// TwinCAT 3 PLC project tmo_motion
// Title: lcls-plc-tmo-motion
// Company: SLAC
// ProjectVersion: 0.0.0
// ProgramVersion: 3.1.4022.7
// CompilerDefines: K
// libraries:
//   LCLS General, * (SLAC)
//   lcls-twincat-common-components, * (SLAC)
//   lcls-twincat-motion, * (SLAC)
//   PMPS, * (SLAC - LCLS)
//   Tc2_MC2, * (Beckhoff Automation GmbH)
//   Tc2_SerialCom, * (Beckhoff Automation GmbH)
//   Tc2_Standard, * (Beckhoff Automation GmbH)
//   Tc2_System, * (Beckhoff Automation GmbH)
//   Tc3_Module, * (Beckhoff Automation GmbH)
// project tree:
//   DUTs/ ENUM_SolidAttenuator_States.TcDUT, ENUM_LaserCoupling_States.TcDUT, ENUM_Sample_Calibration_States.TcDUT, ENUM_ZonePlate_States.TcDUT, E_HomeState.TcDUT
//   GVLs/ GVL_PMPS.TcGVL, GVL_TcGVL.TcGVL, Main.TcGVL
//   / PlcTask.TcTTO (not stored)
//   POUs/ FB_SP_ZP.TcPOU, PRG_1_PlcTask.TcPOU, PRG_2_PMPS_PRE.TcPOU, PRG_3_PMPS_POST.TcPOU, PRG_4_LOG.TcPOU (not stored), PRG_AL1K4_L2SI.TcPOU, PRG_PA1K4_PF.TcPOU, PRG_IM2K4_PPM.TcPOU, PRG_IM3K4_PPM.TcPOU, PRG_IM4K4_PPM.TcPOU, PRG_IM5K4_PPM.TcPOU, PRG_IM6K4_PPM.TcPOU, PRG_LI1K4_IP1.TcPOU, PRG_LI2K4_IP1.TcPOU, PRG_PC5K4.TcPOU, PRG_PF1K4_WFS_TARGET.TcPOU, PRG_PF2K4_WFS_TARGET.TcPOU, PRG_SL1K4_SCATTER.TcPOU, PRG_SP1K4.TcPOU, PRG_ST4K4_TMO_TERM.TcPOU, PRG_ST5K4_TMO_TERM_FIXED.TcPOU, PRG_TM1K4.TcPOU, PRG_TM2K4.TcPOU
//   POUs/Sequence_Mover/ FB_SequenceMover2D.TcPOU
//   POUs/temp/ FB_SLITS.TcPOU, FB_SLITS_POWER.TcPOU, FB_SLITS_SCATTER.TcPOU, FB_ZonePlate_States.TcPOU, PRG_SL2K4_SCATTER.TcPOU
//   POUs/TM1K4/ ENUM_TM1K4_States.TcDUT, FB_TM1K4.TcPOU
//   POUs/TM2K4/ ENUM_TM2K4_States.TcDUT, FB_TM2K4.TcPOU
// real-time tasks:
//   TASK PlcTask: cycle T#10ms, priority 20, ADS port 350
// motion (NC):
//   TASK NC-Task 1 SAF: cycle T#2ms, priority 4, ADS port 501
//   TASK NC-Task 1 SVB: cycle T#10ms, priority 8, ADS port 511
//   AXIS Axis 1 AL1K4-L2SI-MMS (id 1)
//     Dynamic: AccelerationMaximum=200, DecelerationMaximum=200, Acceleration=200, Deceleration=200, Jerk=500, DelayTime=0.004
//     Velo: Maximum=10
//     TargetPosControl: Range=0.002, Time=2
//     OtherSettings: AllowMotionCmdToSlave=true
//     encoder EncType=29
//       EncPara: ScaleFactorNumerator=5e-05, Offset=-214686.941, MaxCount=#xffffffff, ReferenceSystem=1
//         SoftEndMinControl: Enable=true, Range=-108.74
//         SoftEndMaxControl: Enable=true, Range=-30
//         Inc: RefSoftSyncMask=#x0000ffff
//     drive DrvType=24
//       Analog: VeloReferenz=100, ScaleFactorActTorque=0.1
//       TimeComp: TaskDelayCycles=1
//     controller CtrType=2
//       CtrPara: PriorControlFactor=1
//         PosDiffControl: Range=1, Time=0.1
//         PID: PosKp=20, PosExtKp=1, PosExtVelo=0.1, DeadBandPosition=0.002
//         Observer: BandWidth=20
//   AXIS Axis 2 (id 2)
//     OtherSettings: AllowMotionCmdToSlave=true
//     encoder EncType=1
//     drive DrvType=5
//       Analog: ScaleFactorActTorque=0.1
//       TimeComp: TaskDelayCycles=1
//     controller CtrType=1
//       CtrPara: PriorControlFactor=1
//         Observer: BandWidth=20
//   AXIS Axis 3 (id 3)
//     OtherSettings: AllowMotionCmdToSlave=true
//     encoder EncType=1
//     drive DrvType=5
//       Analog: ScaleFactorActTorque=0.1
//       TimeComp: TaskDelayCycles=1
//     controller CtrType=1
//       CtrPara: PriorControlFactor=1
//         Observer: BandWidth=20
//   AXIS Axis 4 (id 4)
//     OtherSettings: AllowMotionCmdToSlave=true
//     encoder EncType=1
//     drive DrvType=5
//       Analog: ScaleFactorActTorque=0.1
//       TimeComp: TaskDelayCycles=1
//     controller CtrType=1
//       CtrPara: PriorControlFactor=1
//         Observer: BandWidth=20
//   AXIS Axis 5 (id 5)
//     OtherSettings: AllowMotionCmdToSlave=true
//     encoder EncType=1
//     drive DrvType=5
//       Analog: ScaleFactorActTorque=0.1
//       TimeComp: TaskDelayCycles=1
//     controller CtrType=1
//       CtrPara: PriorControlFactor=1
//         Observer: BandWidth=20
//   AXIS Axis 6 IM1K4-XTES-MMS (id 6)
//     Velo: Maximum=10
//     OtherSettings: AllowMotionCmdToSlave=true
//     encoder EncType=29
//       EncPara: ScaleFactorNumerator=5e-05, Offset=-398.1892, MaxCount=#x00400000, ReferenceSystem=1
//         SoftEndMinControl: Enable=true, Range=-90
//         SoftEndMaxControl: Enable=true
//         Inc: RefSoftSyncMask=#x00400000
//     drive DrvType=24
//       DrvPara: Inverse=true
//         Analog: VeloReferenz=50, ScaleFactorActTorque=0.1
//         TimeComp: TaskDelayCycles=1
//     controller CtrType=2
//       CtrPara: PriorControlFactor=1
//         PosDiffControl: Range=1
//         PID: PosKp=20, PosExtKp=20, DeadBandPosition=0.001
//         Observer: BandWidth=20
//   AXIS Axis 7 IM1K4-XTES-CLZ (id 7)
//     General: UnitName=%
//     Velo: Maximum=10
//     OtherSettings: AllowMotionCmdToSlave=true
//     encoder EncType=4
//       EncPara: ScaleFactorNumerator=0.003, MaxCount=#x0000ffff
//         SoftEndMinControl: Enable=true, Range=-100
//         SoftEndMaxControl: Enable=true, Range=100
//         Inc: RefSoftSyncMask=#x0000ffff
//     drive DrvType=23
//       DrvPara: Inverse=true
//         Analog: VeloReferenz=33, ScaleFactorActTorque=0.1
//         TimeComp: TaskDelayCycles=1
//     controller CtrType=2
//       CtrPara: PriorControlFactor=1
//         PosDiffControl: Range=1
//         PID: PosKp=20, PosExtKp=20, DeadBandPosition=0.1
//         Observer: BandWidth=20
//   AXIS Axis 8 IM1K4-XTES-CLF (id 8)
//     General: UnitName=%
//     Velo: Maximum=10
//     OtherSettings: AllowMotionCmdToSlave=true
//     encoder EncType=4
//       EncPara: ScaleFactorNumerator=0.008, MaxCount=#x0000ffff
//         SoftEndMinControl: Enable=true, Range=-100
//         SoftEndMaxControl: Enable=true, Range=100
//         Inc: RefSoftSyncMask=#x0000ffff
//     drive DrvType=23
//       DrvPara: Inverse=true
//         Analog: VeloReferenz=70, ScaleFactorActTorque=0.1
//         TimeComp: TaskDelayCycles=1
//     controller CtrType=2
//       CtrPara: PriorControlFactor=1
//         PosDiffControl: Range=1
//         PID: PosKp=20, PosExtKp=20, DeadBandPosition=0.1
//         Observer: BandWidth=20
//   AXIS Axis 9 IM2K4-PPM-MMS (id 9)
//     Dynamic: AccelerationMaximum=200, DecelerationMaximum=200, Acceleration=200, Deceleration=200, Jerk=1000, DelayTime=0.004
//     Velo: Maximum=65
//     MotionControl: Enable=true, Range=0.0005, Time=1
//     TargetPosControl: Range=0.01, Time=1
//     OtherSettings: AllowMotionCmdToSlave=true
//     encoder EncType=29
//       EncPara: ScaleFactorNumerator=5e-05, Offset=-358.0066, MaxCount=#x00400000, ReferenceSystem=1
//         SoftEndMinControl: Enable=true, Range=-100.57
//         SoftEndMaxControl: Enable=true, Range=-7.67
//         Inc: RefSoftSyncMask=#x00400000
//     drive DrvType=24
//       Analog: VeloReferenz=100, ScaleFactorActTorque=0.1
//       TimeComp: TaskDelayCycles=1
//     controller CtrType=2
//       CtrPara: PriorControlFactor=1
//         PosDiffControl: Range=10, Time=0.1
//         PID: PosKp=10, PosExtKp=0.01, PosExtVelo=0.0005, DeadBandPosition=0.0001
//         Observer: BandWidth=20
//   AXIS SL1K4-BOTTOM-M10 (id 10)
//     Velo: RefSearch=0.2, RefSync=0.05, Maximum=2.2
//     OtherSettings: AllowMotionCmdToSlave=true
//     encoder EncType=4
//       EncPara: MaxCount=#x0000ffff
//         SoftEndMinControl: Enable=true, Range=-31.51
//         SoftEndMaxControl: Enable=true
//         Inc: RefSoftSyncMask=#x0000ffff
//     drive DrvType=24
//       Analog: VeloReferenz=2, ScaleFactorActTorque=0.1
//       TimeComp: TaskDelayCycles=1
//     controller CtrType=1
//       CtrPara: PriorControlFactor=1
//         PosDiffControl: Range=0.05
//         Observer: BandWidth=20
//   AXIS SL1K4-TOP-M11 (id 11)
//     Velo: RefSearch=0.2, RefSync=0.05, Maximum=2.2
//     OtherSettings: AllowMotionCmdToSlave=true
//     encoder EncType=4
//       EncPara: Inverse=true, MaxCount=#x0000ffff
//         SoftEndMinControl: Enable=true, Range=-31.99
//         SoftEndMaxControl: Enable=true
//         Inc: RefSoftSyncMask=#x0000ffff
//     drive DrvType=24
//       Analog: VeloReferenz=2, ScaleFactorActTorque=0.1
//       TimeComp: TaskDelayCycles=1
//     controller CtrType=1
//       CtrPara: PriorControlFactor=1
//         PosDiffControl: Range=0.05
//         Observer: BandWidth=20
//   AXIS SL1K4-NORTH-M12 (id 12)
//     Velo: RefSearch=0.2, RefSync=0.05, Maximum=2.2
//     OtherSettings: AllowMotionCmdToSlave=true
//     encoder EncType=4
//       EncPara: Inverse=true, MaxCount=#x0000ffff
//         SoftEndMinControl: Enable=true, Range=-31.5
//         SoftEndMaxControl: Enable=true
//         Inc: RefSoftSyncMask=#x0000ffff
//     drive DrvType=24
//       Analog: VeloReferenz=2, ScaleFactorActTorque=0.1
//       TimeComp: TaskDelayCycles=1
//     controller CtrType=1
//       CtrPara: PriorControlFactor=1
//         PosDiffControl: Range=0.05
//         Observer: BandWidth=20
//   AXIS SL1K4-SOUTH-M13 (id 13)
//     Velo: RefSearch=0.2, RefSync=0.05, Maximum=2.2
//     OtherSettings: AllowMotionCmdToSlave=true
//     encoder EncType=4
//       EncPara: MaxCount=#x0000ffff
//         SoftEndMinControl: Enable=true, Range=-30.29
//         SoftEndMaxControl: Enable=true
//         Inc: RefSoftSyncMask=#x0000ffff
//     drive DrvType=24
//       Analog: VeloReferenz=2, ScaleFactorActTorque=0.1
//       TimeComp: TaskDelayCycles=1
//     controller CtrType=1
//       CtrPara: PriorControlFactor=1
//         PosDiffControl: Range=0.05
//         Observer: BandWidth=20
//   AXIS ST1K4-TEST (id 14)
//     Velo: RefSearch=5, RefSync=5, SlowManual=1, FastManual=5, Maximum=50
//     OtherSettings: AllowMotionCmdToSlave=true
//     encoder EncType=4
//       EncPara: ScaleFactorNumerator=0.000390625, Inverse=true, MaxCount=#x0000ffff
//         Inc: RefSoftSyncMask=#x0000ffff
//     drive DrvType=24
//       DrvPara: Inverse=true
//         Analog: VeloReferenz=50
//         TimeComp: TaskDelayCycles=1
//     controller CtrType=1
//       CtrPara: PriorControlFactor=1
//         PosDiffControl: Enable=false, Range=0.05
//         Observer: BandWidth=20
//   AXIS Axis 15 IM3K4-PPM-MMS (id 15)
//     Dynamic: AccelerationMaximum=200, DecelerationMaximum=200, Acceleration=200, Deceleration=200, Jerk=1000, DelayTime=0.004
//     Velo: Maximum=65
//     MotionControl: Enable=true, Range=0.0005, Time=1
//     TargetPosControl: Range=0.01, Time=1
//     OtherSettings: AllowMotionCmdToSlave=true
//     encoder EncType=29
//       EncPara: ScaleFactorNumerator=5e-05, Offset=-358.0066, MaxCount=#x00400000, ReferenceSystem=1
//         SoftEndMinControl: Enable=true, Range=-97.98
//         SoftEndMaxControl: Enable=true, Range=-5.69
//     drive DrvType=24
//       Analog: VeloReferenz=100, ScaleFactorActTorque=0.1
//       TimeComp: TaskDelayCycles=1
//     controller CtrType=2
//       CtrPara: PriorControlFactor=1
//         PosDiffControl: Range=10, Time=0.1
//         PID: PosKp=10, PosExtKp=0.01, PosExtVelo=0.0005, DeadBandPosition=0.0001
//         Observer: BandWidth=20
//   AXIS Axis 16 IM4K4-PPM-MMS (id 16)
//     Dynamic: AccelerationMaximum=200, DecelerationMaximum=200, Acceleration=200, Deceleration=200, Jerk=1000, DelayTime=0.004
//     Velo: Maximum=65
//     MotionControl: Enable=true, Range=0.0005, Time=1
//     TargetPosControl: Range=0.01, Time=1
//     OtherSettings: AllowMotionCmdToSlave=true
//     encoder EncType=29
//       EncPara: ScaleFactorNumerator=5e-05, Offset=-358.0066, MaxCount=#x00400000, ReferenceSystem=1
//         SoftEndMinControl: Enable=true, Range=-99.53
//         SoftEndMaxControl: Enable=true, Range=-8.43
//     drive DrvType=24
//       Analog: VeloReferenz=100, ScaleFactorActTorque=0.1
//       TimeComp: TaskDelayCycles=1
//     controller CtrType=2
//       CtrPara: PriorControlFactor=1
//         PosDiffControl: Range=10, Time=0.1
//         PID: PosKp=10, PosExtKp=0.01, PosExtVelo=0.0005, DeadBandPosition=0.0001
//         Observer: BandWidth=20
//   AXIS Axis 17 IM5K4-PPM-MMS (id 17)
//     Dynamic: AccelerationMaximum=200, DecelerationMaximum=200, Acceleration=200, Deceleration=200, Jerk=1000, DelayTime=0.004
//     Velo: Maximum=65
//     MotionControl: Enable=true, Range=0.0005, Time=1
//     TargetPosControl: Range=0.01, Time=1
//     OtherSettings: AllowMotionCmdToSlave=true
//     encoder EncType=29
//       EncPara: ScaleFactorNumerator=5e-05, Offset=-358.0066, MaxCount=#x00400000, ReferenceSystem=1
//         SoftEndMinControl: Enable=true, Range=-97.47
//         SoftEndMaxControl: Enable=true, Range=-4.42
//     drive DrvType=24
//       Analog: VeloReferenz=100, ScaleFactorActTorque=0.1
//       TimeComp: TaskDelayCycles=1
//     controller CtrType=2
//       CtrPara: PriorControlFactor=1
//         PosDiffControl: Range=10, Time=0.1
//         PID: PosKp=10, PosExtKp=0.01, PosExtVelo=0.0005, DeadBandPosition=0.0001
//         Observer: BandWidth=20
//   AXIS Axis 18 PF1K4-WFS_TARGET-MMS-Y (id 18)
//     Dynamic: AccelerationMaximum=200, DecelerationMaximum=200, Acceleration=10, Deceleration=10, Jerk=500, DelayTime=0.004
//     Velo: Maximum=20
//     TargetPosControl: Range=0.002, Time=2
//     OtherSettings: AllowMotionCmdToSlave=true
//     encoder EncType=29
//       EncPara: ScaleFactorNumerator=5e-05, Offset=-358.0066, MaxCount=#x00400000, ReferenceSystem=1
//         SoftEndMinControl: Enable=true, Range=-99.33
//         SoftEndMaxControl: Enable=true, Range=-9.97777
//     drive DrvType=24
//       Analog: VeloReferenz=100, ScaleFactorActTorque=0.1
//       TimeComp: TaskDelayCycles=1
//     controller CtrType=2
//       CtrPara: PriorControlFactor=1
//         PosDiffControl: Range=1
//         PID: PosKp=20, PosExtKp=1, PosExtVelo=0.1, DeadBandPosition=0.002
//         Observer: BandWidth=20
//   AXIS Axis 19 PF1K4-WFS_TARGET-MMS-Z (id 19)
//     Dynamic: AccelerationMaximum=200, DecelerationMaximum=200, Acceleration=10, Deceleration=50, Jerk=500
//     Velo: Maximum=5
//     OtherSettings: AllowMotionCmdToSlave=true
//     encoder EncType=29
//       EncPara: ScaleFactorNumerator=5e-05, MaxCount=#xffffffff
//         SoftEndMinControl: Enable=true, Range=12
//         SoftEndMaxControl: Enable=true, Range=54
//         Inc: RefSoftSyncMask=#x0000ffff
//     drive DrvType=24
//       Analog: VeloReferenz=15.875, TorqueSetpointScale=10, ScaleFactorActTorque=0.1
//       TimeComp: TaskDelayCycles=1
//     controller CtrType=1
//       CtrPara: PriorControlFactor=1
//         PosDiffControl: Range=1
//         Observer: BandWidth=20
//   AXIS Axis 20 LI1K4-IP1-MMS (id 20)
//     Dynamic: AccelerationMaximum=200, DecelerationMaximum=200, Acceleration=200, Deceleration=200, Jerk=500, DelayTime=0.004
//     Velo: Maximum=65
//     TargetPosControl: Range=0.002, Time=2
//     OtherSettings: AllowMotionCmdToSlave=true
//     encoder EncType=29
//       EncPara: ScaleFactorNumerator=5e-05, Offset=-358.0066, MaxCount=#x00400000, ReferenceSystem=1
//         SoftEndMinControl: Enable=true, Range=-107.43
//         SoftEndMaxControl: Enable=true, Range=1.35
//     drive DrvType=24
//       Analog: VeloReferenz=100, ScaleFactorActTorque=0.1
//       TimeComp: TaskDelayCycles=1
//     controller CtrType=2
//       CtrPara: PriorControlFactor=1
//         PosDiffControl: Range=1
//         PID: PosKp=20, PosExtKp=1, PosExtVelo=0.1, DeadBandPosition=0.002
//         Observer: BandWidth=20
//   AXIS Axis 21 TM1K4-MMS-Y (id 21)
//     Dynamic: AccelerationMaximum=200, DecelerationMaximum=200, Acceleration=10, Deceleration=10, Jerk=500, DelayTime=0.004
//     Velo: Maximum=20
//     TargetPosControl: Range=0.002, Time=2
//     OtherSettings: AllowMotionCmdToSlave=true
//     encoder EncType=29
//       EncPara: ScaleFactorNumerator=5e-05, Offset=-358.0066, MaxCount=#x00400000, ReferenceSystem=1
//         SoftEndMinControl: Enable=true, Range=-103.65
//         SoftEndMaxControl: Enable=true, Range=1.41
//     drive DrvType=24
//       Analog: VeloReferenz=100, ScaleFactorActTorque=0.1
//       TimeComp: TaskDelayCycles=1
//     controller CtrType=2
//       CtrPara: PriorControlFactor=1
//         PosDiffControl: Enable=false, Range=1
//         PID: PosKp=20, PosExtKp=1, PosExtVelo=0.1, DeadBandPosition=0.002
//         Observer: BandWidth=20
//   AXIS Axis 22 TM1K4-MMS-X (id 22)
//     Dynamic: AccelerationMaximum=200, DecelerationMaximum=200, Acceleration=10, Deceleration=50, Jerk=500
//     Velo: Maximum=5
//     OtherSettings: AllowMotionCmdToSlave=true
//     encoder EncType=29
//       EncPara: ScaleFactorNumerator=5e-05, MaxCount=#xffffffff
//         SoftEndMinControl: Enable=true, Range=12
//         SoftEndMaxControl: Enable=true, Range=54
//         Inc: RefSoftSyncMask=#x0000ffff
//     drive DrvType=24
//       Analog: VeloReferenz=15.875, TorqueSetpointScale=10, ScaleFactorActTorque=0.1
//       TimeComp: TaskDelayCycles=1
//     controller CtrType=1
//       CtrPara: PriorControlFactor=1
//         PosDiffControl: Range=1
//         Observer: BandWidth=20
//   AXIS SL2K4-BOTTOM-M23 (id 23) // C:\Github\lcls-plc-tmo-motion\plc-tmo-motion\_Config\NC\Axes\SL2K4-BOTTOM-M23.xti
//     Velo: RefSearch=0.2, RefSync=0.05, Maximum=2.2
//     OtherSettings: AllowMotionCmdToSlave=true
//     encoder EncType=4
//       EncPara: MaxCount=#x0000ffff
//         SoftEndMinControl: Enable=true, Range=-30.61
//         SoftEndMaxControl: Enable=true
//         Inc: RefSoftSyncMask=#x0000ffff
//     drive DrvType=24
//       Analog: VeloReferenz=2, ScaleFactorActTorque=0.1
//       TimeComp: TaskDelayCycles=1
//     controller CtrType=1
//       CtrPara: PriorControlFactor=1
//         Observer: BandWidth=20
//   AXIS SL2K4-TOP-M24 (id 24) // C:\Github\lcls-plc-tmo-motion\plc-tmo-motion\_Config\NC\Axes\SL2K4-TOP-M24.xti
//     Velo: RefSearch=0.2, RefSync=0.05, Maximum=2.2
//     PositionAreaControl: Range=0.5
//     TargetPosControl: Range=0.1
//     OtherSettings: AllowMotionCmdToSlave=true
//     encoder EncType=4
//       EncPara: Inverse=true, MaxCount=#x0000ffff
//         SoftEndMinControl: Enable=true, Range=-30.91
//         SoftEndMaxControl: Enable=true
//         Inc: RefSoftSyncMask=#x0000ffff
//     drive DrvType=24
//       Analog: VeloReferenz=2, ScaleFactorActTorque=0.1
//       TimeComp: TaskDelayCycles=1
//     controller CtrType=1
//       CtrPara: PriorControlFactor=1
//         PosDiffControl: Range=0.5
//         Observer: BandWidth=20
//   AXIS SL2K4-NORTH-M25 (id 25) // C:\Github\lcls-plc-tmo-motion\plc-tmo-motion\_Config\NC\Axes\SL2K4-NORTH-M25.xti
//     Velo: RefSearch=0.2, RefSync=0.05, Maximum=2.2
//     OtherSettings: AllowMotionCmdToSlave=true
//     encoder EncType=4
//       EncPara: Inverse=true, MaxCount=#x0000ffff
//         SoftEndMinControl: Enable=true, Range=-30.81
//         SoftEndMaxControl: Enable=true
//         Inc: RefSoftSyncMask=#x0000ffff
//     drive DrvType=24
//       Analog: VeloReferenz=2, ScaleFactorActTorque=0.1
//       TimeComp: TaskDelayCycles=1
//     controller CtrType=1
//       CtrPara: PriorControlFactor=1
//         Observer: BandWidth=20
//   AXIS SL2K4-SOUTH-M26 (id 26) // C:\Github\lcls-plc-tmo-motion\plc-tmo-motion\_Config\NC\Axes\SL2K4-SOUTH-M26.xti
//     Velo: RefSearch=0.2, RefSync=0.05, Maximum=2.2
//     OtherSettings: AllowMotionCmdToSlave=true
//     encoder EncType=4
//       EncPara: MaxCount=#x0000ffff
//         SoftEndMinControl: Enable=true, Range=-30.52
//         SoftEndMaxControl: Enable=true
//         Inc: RefSoftSyncMask=#x0000ffff
//     drive DrvType=24
//       Analog: VeloReferenz=2, ScaleFactorActTorque=0.1
//       TimeComp: TaskDelayCycles=1
//     controller CtrType=1
//       CtrPara: PriorControlFactor=1
//         Observer: BandWidth=20
//   AXIS Axis 30 TM2K4-MMS-Y (id 30)
//     Dynamic: AccelerationMaximum=200, DecelerationMaximum=200, Acceleration=10, Deceleration=10, Jerk=500, DelayTime=0.004
//     Velo: Maximum=20
//     TargetPosControl: Range=0.002, Time=2
//     OtherSettings: AllowMotionCmdToSlave=true
//     encoder EncType=29
//       EncPara: ScaleFactorNumerator=5e-05, Offset=-358.0066, MaxCount=#x00400000, ReferenceSystem=1
//         SoftEndMinControl: Enable=true, Range=-103
//         SoftEndMaxControl: Enable=true, Range=2.2
//     drive DrvType=24
//       Analog: VeloReferenz=100, ScaleFactorActTorque=0.1
//       TimeComp: TaskDelayCycles=1
//     controller CtrType=2
//       CtrPara: PriorControlFactor=1
//         PosDiffControl: Range=1
//         PID: PosKp=20, PosExtKp=1, PosExtVelo=0.1, DeadBandPosition=0.002
//         Observer: BandWidth=20
//   AXIS Axis 31 TM2K4-MMS-X (id 31)
//     Dynamic: AccelerationMaximum=200, DecelerationMaximum=200, Acceleration=10, Deceleration=50, Jerk=500
//     Velo: Maximum=5
//     OtherSettings: AllowMotionCmdToSlave=true
//     encoder EncType=29
//       EncPara: ScaleFactorNumerator=5e-05, MaxCount=#x00400000, ReferenceSystem=1
//         SoftEndMinControl: Enable=true, Range=7
//         SoftEndMaxControl: Enable=true, Range=11
//     drive DrvType=24
//       Analog: VeloReferenz=15.875, ScaleFactorActTorque=0.1
//       TimeComp: TaskDelayCycles=1
//     controller CtrType=1
//       CtrPara: PriorControlFactor=1
//         PosDiffControl: Range=0.2
//         Observer: BandWidth=20
//   AXIS Axis 27 IM6K4-PPM-MMS (id 27)
//     Dynamic: AccelerationMaximum=200, DecelerationMaximum=200, Acceleration=200, Deceleration=200, Jerk=500, DelayTime=0.004
//     Velo: Maximum=65
//     TargetPosControl: Range=0.002, Time=2
//     OtherSettings: AllowMotionCmdToSlave=true
//     encoder EncType=29
//       EncPara: ScaleFactorNumerator=5e-05, Offset=-358.0066, MaxCount=#x00400000, ReferenceSystem=1
//         SoftEndMinControl: Enable=true, Range=-97
//         SoftEndMaxControl: Enable=true, Range=-6.5
//     drive DrvType=24
//       Analog: VeloReferenz=100, ScaleFactorActTorque=0.1
//       TimeComp: TaskDelayCycles=1
//     controller CtrType=2
//       CtrPara: PriorControlFactor=1
//         PosDiffControl: Range=10, Time=0.1
//         PID: PosKp=10, PosExtKp=0.01, PosExtVelo=0.0005, DeadBandPosition=0.0001
//         Observer: BandWidth=20
//   AXIS Axis 28 PF2K4-WFS_TARGET-MMS-Y (id 28)
//     Dynamic: AccelerationMaximum=200, DecelerationMaximum=200, Acceleration=10, Deceleration=10, Jerk=500, DelayTime=0.004
//     Velo: Maximum=20
//     TargetPosControl: Range=0.002, Time=2
//     OtherSettings: AllowMotionCmdToSlave=true
//     encoder EncType=29
//       EncPara: ScaleFactorNumerator=5e-05, Offset=-358.065999999999, MaxCount=#x00400000, ReferenceSystem=1
//         SoftEndMinControl: Enable=true, Range=-103
//         SoftEndMaxControl: Enable=true, Range=-9.71
//     drive DrvType=24
//       Analog: VeloReferenz=100, ScaleFactorActTorque=0.1
//       TimeComp: TaskDelayCycles=1
//     controller CtrType=2
//       CtrPara: PriorControlFactor=1
//         PosDiffControl: Range=1
//         PID: PosKp=20, PosExtKp=1, PosExtVelo=0.1, DeadBandPosition=0.002
//         Observer: BandWidth=20
//   AXIS Axis 29 PF2K4-WFS_TARGET-MMS-Z (id 29)
//     Dynamic: AccelerationMaximum=200, DecelerationMaximum=200, Acceleration=10, Deceleration=50, Jerk=500
//     Velo: Maximum=5
//     OtherSettings: AllowMotionCmdToSlave=true
//     encoder EncType=29
//       EncPara: ScaleFactorNumerator=5e-05, MaxCount=#x00400000, ReferenceSystem=1
//         SoftEndMinControl: Enable=true, Range=17
//         SoftEndMaxControl: Enable=true, Range=50
//     drive DrvType=24
//       DrvPara: Inverse=true
//         Analog: VeloReferenz=15.875, ScaleFactorActTorque=0.1
//         TimeComp: TaskDelayCycles=1
//     controller CtrType=1
//       CtrPara: PriorControlFactor=1
//         PosDiffControl: Range=1
//         Observer: BandWidth=20
//   AXIS LensX (id 32)
//     Dynamic: Acceleration=2, Deceleration=2
//     Velo: SlowManual=0.1, FastManual=1, Maximum=1
//     OtherSettings: AllowMotionCmdToSlave=true, PulseDistancePos=0.5, PulseDistanceNeg=0.5
//     encoder EncType=4
//       EncPara: ScaleFactorNumerator=3.90625e-05, MaxCount=#x0000ffff
//         Inc: RefSoftSyncMask=#x0000ffff
//     drive DrvType=24
//       Analog: VeloReferenz=4.5, ScaleFactorActTorque=0.1
//       TimeComp: TaskDelayCycles=1
//     controller CtrType=2
//       CtrPara: PriorControlFactor=1
//         PosDiffControl: Range=1
//         Observer: BandWidth=20
//   AXIS FoilX (id 33)
//     Dynamic: Acceleration=2, Deceleration=2
//     Velo: SlowManual=0.1, FastManual=1, Maximum=27
//     PositionAreaControl: Range=0.1
//     TargetPosControl: Range=0.1
//     OtherSettings: AllowMotionCmdToSlave=true, PulseDistancePos=0.5, PulseDistanceNeg=0.5
//     encoder EncType=29
//       EncPara: ScaleFactorNumerator=5e-05, MaxCount=#xffffffff
//         Inc: RefSoftSyncMask=#x0000ffff
//     drive DrvType=24
//       DrvPara: Inverse=true
//         Analog: VeloReferenz=25.4, ScaleFactorActTorque=0.1
//         TimeComp: TaskDelayCycles=1
//     controller CtrType=2
//       CtrPara: PriorControlFactor=1
//         PosDiffControl: Range=0.8
//         Observer: BandWidth=20
//   AXIS ZonePlateX (id 34)
//     Dynamic: Acceleration=2, Deceleration=2
//     Velo: SlowManual=0.1, FastManual=1, Maximum=5
//     TargetPosControl: Range=0.03, Time=0.1
//     OtherSettings: AllowMotionCmdToSlave=true, PulseDistancePos=0.5, PulseDistanceNeg=0.5
//     encoder EncType=29
//       EncPara: ScaleFactorNumerator=5e-05, MaxCount=#xffffffff
//         SoftEndMinControl: Enable=true
//         SoftEndMaxControl: Enable=true, Range=125.6
//         Inc: RefSoftSyncMask=#x0000ffff
//     drive DrvType=24
//       DrvPara: Inverse=true
//         Analog: VeloReferenz=13.2, ScaleFactorActTorque=0.1
//         TimeComp: TaskDelayCycles=1
//     controller CtrType=2
//       CtrPara: PriorControlFactor=1
//         PosDiffControl: Range=1
//         PID: PosKp=2
//         Observer: BandWidth=20
//   AXIS ZonePlateY (id 35)
//     Dynamic: Acceleration=2, Deceleration=2
//     Velo: SlowManual=0.1, FastManual=1, Maximum=5
//     OtherSettings: AllowMotionCmdToSlave=true, PulseDistancePos=0.5, PulseDistanceNeg=0.5
//     encoder EncType=29
//       EncPara: ScaleFactorNumerator=5e-05, Offset=-214733.3875, MaxCount=#xffffffff
//         SoftEndMinControl: Enable=true, Range=-10.6
//         SoftEndMaxControl: Enable=true, Range=3.8
//         Inc: RefSoftSyncMask=#x0000ffff
//     drive DrvType=24
//       Analog: VeloReferenz=6, ScaleFactorActTorque=0.1
//       TimeComp: TaskDelayCycles=1
//     controller CtrType=2
//       CtrPara: PriorControlFactor=1
//         PosDiffControl: Range=0.8, Time=0.1
//         Observer: BandWidth=20
//   AXIS ZonePlateZ (id 36)
//     Dynamic: Acceleration=2, Deceleration=2
//     Velo: SlowManual=0.1, FastManual=1, Maximum=5
//     TargetPosControl: Range=0.3
//     OtherSettings: AllowMotionCmdToSlave=true, PulseDistancePos=0.5, PulseDistanceNeg=0.5
//     encoder EncType=29
//       EncPara: ScaleFactorNumerator=5e-05, ScaleFactorDenominator=1.6, Offset=-134207.665, MaxCount=#xffffffff
//         SoftEndMinControl: Enable=true, Range=-1
//         SoftEndMaxControl: Enable=true, Range=2
//         Inc: RefSoftSyncMask=#x0000ffff
//     drive DrvType=24
//       Analog: VeloReferenz=6.25, ScaleFactorActTorque=0.1
//       TimeComp: TaskDelayCycles=1
//     controller CtrType=2
//       CtrPara: PriorControlFactor=1
//         PosDiffControl: Range=1
//         Observer: BandWidth=20
//   AXIS YagX (id 37)
//     Dynamic: Acceleration=2, Deceleration=2
//     Velo: SlowManual=0.1, FastManual=1, Maximum=1
//     OtherSettings: AllowMotionCmdToSlave=true, PulseDistancePos=0.5, PulseDistanceNeg=0.5
//     encoder EncType=29
//       EncPara: ScaleFactorNumerator=5e-05, Offset=128, Inverse=true, MaxCount=#xffffffff, MaxCountHighDWord=#x0000001f
//         Inc: RefSoftSyncMask=#x0000ffff
//     drive DrvType=24
//       Analog: VeloReferenz=10, ScaleFactorActTorque=0.1
//       TimeComp: TaskDelayCycles=1
//     controller CtrType=2
//       CtrPara: PriorControlFactor=1
//         PosDiffControl: Range=1
//         Observer: BandWidth=20
//   AXIS YagY (id 38)
//     Dynamic: Acceleration=2, Deceleration=2
//     Velo: SlowManual=0.1, FastManual=1, Maximum=1
//     OtherSettings: AllowMotionCmdToSlave=true, PulseDistancePos=0.5, PulseDistanceNeg=0.5
//     encoder EncType=4
//       EncPara: ScaleFactorNumerator=7.8125e-05, MaxCount=#x0000ffff
//         Inc: RefSoftSyncMask=#x0000ffff
//     drive DrvType=24
//       Analog: VeloReferenz=10, ScaleFactorActTorque=0.1
//       TimeComp: TaskDelayCycles=1
//     controller CtrType=2
//       CtrPara: PriorControlFactor=1
//         PosDiffControl: Range=1
//         Observer: BandWidth=20
//   AXIS YagZ (id 39)
//     Dynamic: Acceleration=2, Deceleration=2
//     Velo: SlowManual=0.1, FastManual=1, Maximum=1
//     OtherSettings: AllowMotionCmdToSlave=true, PulseDistancePos=0.5, PulseDistanceNeg=0.5
//     encoder EncType=29
//       EncPara: ScaleFactorNumerator=5e-05, Offset=172, Inverse=true, MaxCount=#xffffffff, MaxCountHighDWord=#x0000001f
//         Inc: RefSoftSyncMask=#x0000ffff
//     drive DrvType=24
//       Analog: VeloReferenz=12.7, ScaleFactorActTorque=0.1
//       TimeComp: TaskDelayCycles=1
//     controller CtrType=2
//       CtrPara: PriorControlFactor=1
//         PosDiffControl: Range=1
//         Observer: BandWidth=20
//   AXIS YagTheta (id 40)
//     Dynamic: Acceleration=2, Deceleration=2
//     Velo: SlowManual=0.1, FastManual=1, Maximum=1
//     TargetPosControl: Range=0.001, Time=0.8
//     OtherSettings: AllowMotionCmdToSlave=true, PulseDistancePos=0.5, PulseDistanceNeg=0.5
//     encoder EncType=4
//       EncPara: ScaleFactorNumerator=1.171875e-05, ScaleFactorDenominator=0.036667, MaxCount=#x0000ffff
//         Inc: RefSoftSyncMask=#x0000ffff
//     drive DrvType=24
//       Analog: VeloReferenz=409.0905372, ScaleFactorActTorque=0.1
//       TimeComp: TaskDelayCycles=1
//     controller CtrType=2
//       CtrPara: PriorControlFactor=1
//         PosDiffControl: Range=1
//         PID: PosKp=5, DeadBandPosition=0.001
//         Observer: BandWidth=20
//   AXIS Thorlabs1 (id 41)
//     Dynamic: AccelerationMaximum=10, DecelerationMaximum=10, Acceleration=5, Deceleration=5
//     Velo: Maximum=2
//     OtherSettings: AllowMotionCmdToSlave=true
//     encoder EncType=4
//       EncPara: ScaleFactorNumerator=1.593130056e-05, MaxCount=#x0000ffff
//         Inc: RefSoftSyncMask=#x0000ffff
//     drive DrvType=24
//       Analog: VeloReferenz=2.039206472, ScaleFactorActTorque=0.1
//       TimeComp: TaskDelayCycles=1
//     controller CtrType=1
//       CtrPara: PriorControlFactor=1
//         PID: PosKp=0
//         Observer: BandWidth=20
//   AXIS Thorlabs2 (id 42)
//     Dynamic: AccelerationMaximum=10, DecelerationMaximum=10, Acceleration=5, Deceleration=5
//     Velo: Maximum=2
//     OtherSettings: AllowMotionCmdToSlave=true
//     encoder EncType=4
//       EncPara: ScaleFactorNumerator=1.593130056e-05, MaxCount=#x0000ffff
//         Inc: RefSoftSyncMask=#x0000ffff
//     drive DrvType=24
//       Analog: VeloReferenz=2.039206472, ScaleFactorActTorque=0.1
//       TimeComp: TaskDelayCycles=1
//     controller CtrType=1
//       CtrPara: PriorControlFactor=1
//         PID: PosKp=0
//         Observer: BandWidth=20
//   AXIS Thorlab-LenX (id 43)
//     Velo: Maximum=15
//     PositionAreaControl: Range=0.1
//     OtherSettings: AllowMotionCmdToSlave=true
//     encoder EncType=29
//       EncPara: ScaleFactorNumerator=5e-05, MaxCount=#xffffffff, MaxCountHighDWord=#x0000001f
//         Inc: RefSoftSyncMask=#x0000ffff
//     drive DrvType=24
//       Analog: VeloReferenz=10, ScaleFactorActTorque=0.1
//       TimeComp: TaskDelayCycles=1
//     controller CtrType=1
//       CtrPara: PriorControlFactor=1
//         PosDiffControl: Range=0.1
//         Observer: BandWidth=20
//   AXIS FoilY (id 44)
//     Velo: Maximum=7
//     PositionAreaControl: Range=0.1
//     OtherSettings: AllowMotionCmdToSlave=true
//     encoder EncType=29
//       EncPara: ScaleFactorNumerator=5e-05, Offset=-214725.8336, MaxCount=#xffffffff
//         Inc: RefSoftSyncMask=#x0000ffff
//     drive DrvType=24
//       Analog: VeloReferenz=5.08, ScaleFactorActTorque=0.1
//       TimeComp: TaskDelayCycles=1
//     controller CtrType=1
//       CtrPara: PriorControlFactor=1
//         PosDiffControl: Range=0.8
//         Observer: BandWidth=20
//   AXIS Axis 45 LI2K4-MMS-Y (id 45)
//     Dynamic: Acceleration=2, Deceleration=2
//     Velo: RefSearch=0.1, RefSync=0.1, SlowManual=0.1, FastManual=0.1, Maximum=5
//     PositionAreaControl: Range=0.05
//     TargetPosControl: Range=0.1
//     OtherSettings: AllowMotionCmdToSlave=true, PulseDistancePos=0.1, PulseDistanceNeg=0.1
//     encoder EncType=29
//       EncPara: ScaleFactorNumerator=5e-05, Offset=-214569.724, MaxCount=#xffffffff
//         Inc: RefSoftSyncMask=#x0000ffff
//     drive DrvType=24
//       Analog: VeloReferenz=20.9, ScaleFactorActTorque=0.1
//       TimeComp: TaskDelayCycles=1
//     controller CtrType=2
//       CtrPara: PriorControlFactor=1
//         PosDiffControl: Range=0.8, Time=0.1
//         PID: DeadBandPosition=0.1
//         Observer: BandWidth=20
//   AXIS Axis 46 LI2K4-MMS-X (id 46)
//     Velo: RefSearch=0.1, RefSync=0.1, SlowManual=0.1, FastManual=0.1, Maximum=5
//     PositionAreaControl: Range=0.1
//     OtherSettings: AllowMotionCmdToSlave=true, PulseDistancePos=0.1, PulseDistanceNeg=0.1
//     encoder EncType=29
//       EncPara: ScaleFactorNumerator=5e-05, Offset=-214728.674, MaxCount=#xffffffff
//         SoftEndMinControl: Range=-4
//         SoftEndMaxControl: Range=1.5
//         Inc: RefSoftSyncMask=#x0000ffff
//     drive DrvType=24
//       DrvPara: Inverse=true
//         Analog: VeloReferenz=6.1, ScaleFactorActTorque=0.1
//         TimeComp: TaskDelayCycles=1
//     controller CtrType=2
//       CtrPara: PriorControlFactor=1
//         PosDiffControl: Range=0.8
//         PID: DeadBandPosition=0.1
//         Observer: BandWidth=20
//   AXIS PA1K4-PF-MMS (id 47)
//     Velo: Maximum=7
//     PositionAreaControl: Range=0.1
//     OtherSettings: AllowMotionCmdToSlave=true
//     encoder EncType=29
//       EncPara: ScaleFactorNumerator=5e-05, MaxCount=#xffffffff
//         SoftEndMinControl: Enable=true, Range=39
//         SoftEndMaxControl: Enable=true, Range=182.5
//         Inc: RefSoftSyncMask=#x0000ffff
//     drive DrvType=24
//       Analog: VeloReferenz=20.9, ScaleFactorActTorque=0.1
//       TimeComp: TaskDelayCycles=1
//     controller CtrType=1
//       CtrPara: PriorControlFactor=1
//         PosDiffControl: Range=0.9, Time=0.1
//         Observer: BandWidth=20
// I/O:
//   DEVICE Device 1 (EtherCAT), AmsNetId 0.0.0.0.2.1
//     Power (EK1200) [EK1200-5000 EtherCAT Power supply (2A E-Bus)]
//       PMPS FFO (EL2202)
//       License (EL6070) [EL6070 1Ch. Licensing-Terminal] (disabled)
//       PMPS_Bridge (EL6692) [EL6692 EtherCAT Bridge terminal (Primary)]
//       PLC Junction 1 (EK1122) [EK1122 2 port EtherCAT junction] (disabled)
//         X1 TMO FEE EC1 (EK1100) [EK1100 EtherCAT Coupler (2A E-Bus)] (disabled)
//           FEE EC1 E1 (EK1122) [EK1122 2 port EtherCAT junction]
//             X1 IM1K4-XTES (EK1100) [EK1100 EtherCAT Coupler (2A E-Bus)] (disabled)
//               IM1K4-EL7041-E1 [EL7041 1Ch. Stepper motor output stage (50V, 5A)]
//               IM1K4-EL2004-E2 [EL2004 4Ch. Dig. Output 24V, 0.5A]
//               IM1K4-EL5042-E3 [EL5042 2Ch. BiSS-C Encoder]
//               IM1K4-EL7342-E4 [EL7342 2Ch. DC motor output stage (50V, 3.5A)]
//               IM1K4-EL1088-E5 [EL1088 8Ch. Dig. Input 24V, 3ms, negative]
//               IM1K4-EL6002-E6 [EL6002 Interface 2Ch. (RS232)]
//               IM1K4-EL9011 [EL9011 End Terminal]
//             X2-ST1K4-TEST (EK1100) [EK1100 EtherCAT Coupler (2A E-Bus)] (disabled)
//               ST1K4-EL3314-E1 [EL3314 4Ch. Ana. Input Thermocouple (TC)]
//               ST1K4-EL3142-E2 [EL3142 2Ch. Ana Input 0-20mA]
//               ST1K4-EL2202-E3 [EL2202 2Ch. Dig. Output 24V, 0.5A]
//               ST1K4-EL7041-E4 [EL7041 1Ch. Stepper motor output stage (50V, 5A)]
//               ST1K4-EL9505-E5 [EL9505 Power supply terminal 5V]
//               ST1K4-EL9011 [EL9011 End Terminal]
//           FEE EC1 E2 (EK1122) [EK1122 2 port EtherCAT junction]
//             X1 AT1K4-SOLID (EK1100) [EK1100 EtherCAT Coupler (2A E-Bus)]
//               AT1K4-EL7047-01 [EL7047 1Ch. Stepper motor output stage (50V, 5A)]
//               AT1K4-EL7047-02 [EL7047 1Ch. Stepper motor output stage (50V, 5A)]
//               AT1K4-EL7047-03 [EL7047 1Ch. Stepper motor output stage (50V, 5A)]
//               AT1K4-EL7047-04 [EL7047 1Ch. Stepper motor output stage (50V, 5A)]
//               AT1K4-EL5042-01 [EL5042 2Ch. BiSS-C Encoder]
//               AT1K4-EL5042-02 [EL5042 2Ch. BiSS-C Encoder]
//               AT1K4-EL3202-01 [EL3202-0020 2Ch. Ana. Input PT100 (RTD), High Precision, calibrated]
//               AT1K4-EL3202-02 [EL3202-0020 2Ch. Ana. Input PT100 (RTD), High Precision, calibrated]
//               AT1K4-EL3202-03 [EL3202-0020 2Ch. Ana. Input PT100 (RTD), High Precision, calibrated]
//               AT1K4-EL3202-04 [EL3202-0020 2Ch. Ana. Input PT100 (RTD), High Precision, calibrated]
//               Term 119 (EL9011) [EL9011 End Terminal]
//           FEE EC1 End Cap (EL9011)
//         X2 TMO FEE EC2 (EK1100)
//       PLC Junction 2 (EK1122) [EK1122 2 port EtherCAT junction]
//         PLC Coupler 1(EK1100)
//         PLC Coupler 2 (EK1100) [EK1100 EtherCAT Coupler (2A E-Bus)]
//           PLC Junction 7 (EK1122) [EK1122 2 port EtherCAT junction]
//             LI3K4-LIC (EK1100) [EK1100 EtherCAT Coupler (2A E-Bus)] (disabled)
//             TM1K4-ATM (EK1100) [EK1100 EtherCAT Coupler (2A E-Bus)]
//               TM1K4-EL7041-1
//               TM1K4-EL7041-2
//               TM1K4-EL5042
//               TM1K4-EL2004
//               TM1K4-EL3314
//               TM1K4-EL9011
//           PLC Junction 8 (EK1122) [EK1122 2 port EtherCAT junction]
//             IM5K4-PPM (EK1100) [EK1100 EtherCAT Coupler (2A E-Bus)]
//               IM5K4-EL7041-E1 [EL7041 1Ch. Stepper motor output stage (50V, 5A)]
//               IM5K4-EL5042-E2 [EL5042 2Ch. BiSS-C Encoder]
//               IM5K4-EL2004-E3 [EL2004 4Ch. Dig. Output 24V, 0.5A]
//               IM5K4-EL3314-E4 [EL3314 4Ch. Ana. Input Thermocouple (TC)]
//               IM5K4-EL3052-E5 [EL3052 2Ch. Ana. Input 4-20mA]
//               IM5K4-EL3062-E6 [EL3062 2Ch. Ana. Input 0-10V]
//               IM5K4-EL4004-E7 [EL4004 4Ch. Ana. Output 0-10V, 12bit]
//               IM5K4-EL9011 [EL9011 End Terminal]
//             ST4K4-TERM (EP2338-0001) [EP2338-0001 8 Ch. Dig. Input/Output 24V, 0,5A, M8]
//             EP3174-FWM-E2 [EP3174-0002 4Ch. Ana. Input +/-10V, 0-10V, 0/4-20mA configurable]
//           PLC Junction 9 (EK1122) [EK1122 2 port EtherCAT junction]
//             X2 SL2K4-SCATTER [EK1100 EtherCAT Coupler (2A E-Bus)] (disabled)
//               SL2K4-EL7031-E1 [EL7031 1Ch. Stepper motor output stage (24V, 1.5A)]
//               SL2K4-EL5101-E2 [EL5101 1Ch. Inc. Encoder 5V]
//               SL2K4-EL7031-E3 [EL7031 1Ch. Stepper motor output stage (24V, 1.5A)]
//               SL2K4-EL5101-E4 [EL5101 1Ch. Inc. Encoder 5V]
//               SL2K4-EL7031-E5 [EL7031 1Ch. Stepper motor output stage (24V, 1.5A)]
//               SL2K4-EL5101-E6 [EL5101 1Ch. Inc. Encoder 5V]
//               SL2K4-EL7031-E7 [EL7031 1Ch. Stepper motor output stage (24V, 1.5A)]
//               SL2K4-EL5101-E8 [EL5101 1Ch. Inc. Encoder 5V]
//               SL2K4-EL9011
//             LI2K4-PA1K4 (EK1100) [EK1100 EtherCAT Coupler (2A E-Bus)]
//               LI2K4Y-EL7047-E1 [EL7047 1Ch. Stepper motor output stage (50V, 5A)]
//               LI2K4-EL5042-E2
//               LI2K4X-EL7047-E3
//               PA1K4-PF-EL7047-E4 [EL7047 1Ch. Stepper motor output stage (50V, 5A)]
//               PA1K4-PF-EL5042-E5 [EL5042 2Ch. BiSS-C Encoder]
//               Term 323 (EL9011)
//             SP1K4 Top Rail (EK1100) [EK1100 EtherCAT Coupler (2A E-Bus)]
//               SP1K4-EL5042-E1 [EL5042 2Ch. BiSS-C Encoder]
//               SP1K4-EL5042-E2 [EL5042 2Ch. BiSS-C Encoder]
//               Term 9 (EL7041) [EL7041 1Ch. Stepper motor output stage (50V, 5A)]
//               Term 10 (EL7041) [EL7041 1Ch. Stepper motor output stage (50V, 5A)]
//               FoilY-EL7041 [EL7041 1Ch. Stepper motor output stage (50V, 5A)]
//               Thorlab-LenX-EL7031 [EL7031 1Ch. Stepper motor output stage (24V, 1.5A)]
//               SP1K4-EL5042-E7 [EL5042 2Ch. BiSS-C Encoder]
//               SP1K4-EL5042-E8 [EL5042 2Ch. BiSS-C Encoder]
//               SP1K4-EL5042-E9 [EL5042 2Ch. BiSS-C Encoder]
//               Term 11 (EL9505) [EL9505 Power supply terminal 5V]
//               SP1K4-TL1-EL1124 [EL1124 4Ch. Dig. Input 5V, 10µs, Sensor Power]
//               Term 13 (EL9505) [EL9505 Power supply terminal 5V]
//               SP1K4-TL2-EL1124 [EL1124 4Ch. Dig. Input 5V, 10µs, Sensor Power]
//               SP1K4-EL3202-E9A
//               SP1K4-EL3202-E9B [EL3202-0010 2Ch. Ana. Input PT100 (RTD), High Precision]
//               Term 15 (EK1122) [EK1122 2 port EtherCAT junction]
//               Term 300 (EL9011) [EL9011 End Terminal]
//             SP1K4 Bottom Rail (EK1100) [EK1100 EtherCAT Coupler (2A E-Bus)]
//               EL7031-LensX [EL7031 1Ch. Stepper motor output stage (24V, 1.5A)]
//               LensX_EL1004 [EL1004 4Ch. Dig. Input 24V, 3ms]
//               FoilX-EL7041 [EL7041 1Ch. Stepper motor output stage (50V, 5A)]
//               ZonePlateX-EL7041 [EL7041 1Ch. Stepper motor output stage (50V, 5A)]
//               ZonePlateY-EL7041 [EL7041 1Ch. Stepper motor output stage (50V, 5A)]
//               ZonePlateZ-EL7041 [EL7041 1Ch. Stepper motor output stage (50V, 5A)]
//               YagX-EL7041 [EL7041 1Ch. Stepper motor output stage (50V, 5A)]
//               YagY-EL7041 [EL7041 1Ch. Stepper motor output stage (50V, 5A)]
//               YagZ-EL7041 [EL7041 1Ch. Stepper motor output stage (50V, 5A)]
//               YagTheta-EL7041 [EL7041 1Ch. Stepper motor output stage (50V, 5A)]
//               Term 301 (EL9011) [EL9011 End Terminal]
//           PLC Junction 10 (EK1122) [EK1122 2 port EtherCAT junction]
//             Term 201 (EK1100) [EK1100 EtherCAT Coupler (2A E-Bus)]
//               Term 202 (EL7041)
//               Term 203 (EL7041)
//               Term 204 (EL5042) [EL5042 2Ch. BiSS-C Encoder]
//               Term 205 (EL2004) [EL2004 4Ch. Dig. Output 24V, 0.5A]
//               Term 206 (EL3314) [EL3314 4Ch. Ana. Input Thermocouple (TC)]
//               Term 221 (EL9011)
//       PLC Junction 3 (EK1122) [EK1122 2 port EtherCAT junction] (disabled)
//       PLC Junction 4 (EK1122) [EK1122 2 port EtherCAT junction] (disabled)
//       PLC End Coupler (EK1110) [EK1110 EtherCAT extension]
// variable links:
//   Axes/SL1K4-BOTTOM-M10 <-> Device 1 (EtherCAT)/Power (EK1200)/PLC Junction 1 (EK1122)/X2 TMO FEE EC2 (EK1100)/FEE EC2 E1 (EK1122)/X2 SL1K4-SCATTER/SL1K4-EL5101-E2
//     Enc/Inputs/In/nDataIn1[0] <-> ENC Status compact/Counter value
//     Enc/Inputs/In/nDataIn2[0] <-> ENC Status compact/Latch value
//     Enc/Inputs/In/nState1 @bit 4 <-> ENC Status compact/Status/Counter overflow
//     Enc/Inputs/In/nState1 @bit 3 <-> ENC Status compact/Status/Counter underflow
//     Enc/Inputs/In/nState1 @bit 7 <-> ENC Status compact/Status/Extrapolation stall
//     Enc/Inputs/In/nState1 <-> ENC Status compact/Status/Latch C valid
//     Enc/Inputs/In/nState1 @bit 1 <-> ENC Status compact/Status/Latch extern valid
//     Enc/Inputs/In/nState1 @bit 6 <-> ENC Status compact/Status/Open circuit
//     Enc/Inputs/In/nState1 @bit 2 <-> ENC Status compact/Status/Set counter done
//     Enc/Inputs/In/nState1 @bit 5 <-> ENC Status compact/Status/Status of input status
//     Enc/Inputs/In/nState2 @bit 4 <-> ENC Status compact/Status/Status of extern latch
//     Enc/Inputs/In/nState2 <-> ENC Status compact/Status/Status of input A
//     Enc/Inputs/In/nState2 @bit 1 <-> ENC Status compact/Status/Status of input B
//     Enc/Inputs/In/nState2 @bit 2 <-> ENC Status compact/Status/Status of input C
//     Enc/Inputs/In/nState2 @bit 3 <-> ENC Status compact/Status/Status of input gate
//     Enc/Inputs/In/nState2 @bit 5 <-> ENC Status compact/Status/Sync error
//     Enc/Inputs/In/nState2 @bit 6 <-> ENC Status compact/Status/TxPDO State
//     Enc/Inputs/In/nState2 @bit 7 <-> ENC Status compact/Status/TxPDO Toggle
//     Enc/Inputs/In/nState4 @bit 1 <-> WcState/InputToggle
//     Enc/Inputs/In/nState4 <-> WcState/WcState
//     Enc/Outputs/Out/nCtrl1 <-> ENC Control compact/Control/Enable latch C
//     Enc/Outputs/Out/nCtrl1 @bit 3 <-> ENC Control compact/Control/Enable latch extern on negative edge
//     Enc/Outputs/Out/nCtrl1 @bit 1 <-> ENC Control compact/Control/Enable latch extern on positive edge
//     Enc/Outputs/Out/nCtrl1 @bit 2 <-> ENC Control compact/Control/Set counter
//     Enc/Outputs/Out/nDataOut1[0] <-> ENC Control compact/Set counter value
//   Axes/SL1K4-BOTTOM-M10 <-> Device 1 (EtherCAT)/Power (EK1200)/PLC Junction 1 (EK1122)/X2 TMO FEE EC2 (EK1100)/FEE EC2 E1 (EK1122)/X2 SL1K4-SCATTER/SL1K4-EL7031-E1
//     Drive/Inputs/In/nState1 @bit 3 <-> STM Status/Status/Error
//     Drive/Inputs/In/nState1 @bit 5 <-> STM Status/Status/Moving negative
//     Drive/Inputs/In/nState1 @bit 4 <-> STM Status/Status/Moving positive
//     Drive/Inputs/In/nState1 @bit 1 <-> STM Status/Status/Ready
//     Drive/Inputs/In/nState1 <-> STM Status/Status/Ready to enable
//     Drive/Inputs/In/nState1 @bit 6 <-> STM Status/Status/Torque reduced
//     Drive/Inputs/In/nState1 @bit 2 <-> STM Status/Status/Warning
//     Drive/Inputs/In/nState2 @bit 3 <-> STM Status/Status/Digital input 1
//     Drive/Inputs/In/nState2 @bit 4 <-> STM Status/Status/Digital input 2
//     Drive/Inputs/In/nState2 @bit 5 <-> STM Status/Status/Sync error
//     Drive/Inputs/In/nState2 @bit 7 <-> STM Status/Status/TxPDO Toggle
//     Drive/Inputs/In/nState4 @bit 1 <-> WcState/InputToggle
//     Drive/Inputs/In/nState4 <-> WcState/WcState
//     Drive/Outputs/Out/nCtrl1 <-> STM Control/Control/Enable
//     Drive/Outputs/Out/nCtrl1 @bit 2 <-> STM Control/Control/Reduce torque
//     Drive/Outputs/Out/nCtrl1 @bit 1 <-> STM Control/Control/Reset
//     Drive/Outputs/Out/nDataOut2[0] <-> STM Velocity/Velocity
//   Axes/SL1K4-NORTH-M12 <-> Device 1 (EtherCAT)/Power (EK1200)/PLC Junction 1 (EK1122)/X2 TMO FEE EC2 (EK1100)/FEE EC2 E1 (EK1122)/X2 SL1K4-SCATTER/SL1K4-EL5101-E6
//     Enc/Inputs/In/nDataIn1[0] <-> ENC Status compact/Counter value
//     Enc/Inputs/In/nDataIn2[0] <-> ENC Status compact/Latch value
//     Enc/Inputs/In/nState1 @bit 4 <-> ENC Status compact/Status/Counter overflow
//     Enc/Inputs/In/nState1 @bit 3 <-> ENC Status compact/Status/Counter underflow
//     Enc/Inputs/In/nState1 @bit 7 <-> ENC Status compact/Status/Extrapolation stall
//     Enc/Inputs/In/nState1 <-> ENC Status compact/Status/Latch C valid
//     Enc/Inputs/In/nState1 @bit 1 <-> ENC Status compact/Status/Latch extern valid
//     Enc/Inputs/In/nState1 @bit 6 <-> ENC Status compact/Status/Open circuit
//     Enc/Inputs/In/nState1 @bit 2 <-> ENC Status compact/Status/Set counter done
//     Enc/Inputs/In/nState1 @bit 5 <-> ENC Status compact/Status/Status of input status
//     Enc/Inputs/In/nState2 @bit 4 <-> ENC Status compact/Status/Status of extern latch
//     Enc/Inputs/In/nState2 <-> ENC Status compact/Status/Status of input A
//     Enc/Inputs/In/nState2 @bit 1 <-> ENC Status compact/Status/Status of input B
//     Enc/Inputs/In/nState2 @bit 2 <-> ENC Status compact/Status/Status of input C
//     Enc/Inputs/In/nState2 @bit 3 <-> ENC Status compact/Status/Status of input gate
//     Enc/Inputs/In/nState2 @bit 5 <-> ENC Status compact/Status/Sync error
//     Enc/Inputs/In/nState2 @bit 6 <-> ENC Status compact/Status/TxPDO State
//     Enc/Inputs/In/nState2 @bit 7 <-> ENC Status compact/Status/TxPDO Toggle
//     Enc/Inputs/In/nState4 @bit 1 <-> WcState/InputToggle
//     Enc/Inputs/In/nState4 <-> WcState/WcState
//     Enc/Outputs/Out/nCtrl1 <-> ENC Control compact/Control/Enable latch C
//     Enc/Outputs/Out/nCtrl1 @bit 3 <-> ENC Control compact/Control/Enable latch extern on negative edge
//     Enc/Outputs/Out/nCtrl1 @bit 1 <-> ENC Control compact/Control/Enable latch extern on positive edge
//     Enc/Outputs/Out/nCtrl1 @bit 2 <-> ENC Control compact/Control/Set counter
//     Enc/Outputs/Out/nDataOut1[0] <-> ENC Control compact/Set counter value
//   Axes/SL1K4-NORTH-M12 <-> Device 1 (EtherCAT)/Power (EK1200)/PLC Junction 1 (EK1122)/X2 TMO FEE EC2 (EK1100)/FEE EC2 E1 (EK1122)/X2 SL1K4-SCATTER/SL1K4-EL7031-E5
//     Drive/Inputs/In/nState1 @bit 3 <-> STM Status/Status/Error
//     Drive/Inputs/In/nState1 @bit 5 <-> STM Status/Status/Moving negative
//     Drive/Inputs/In/nState1 @bit 4 <-> STM Status/Status/Moving positive
//     Drive/Inputs/In/nState1 @bit 1 <-> STM Status/Status/Ready
//     Drive/Inputs/In/nState1 <-> STM Status/Status/Ready to enable
//     Drive/Inputs/In/nState1 @bit 6 <-> STM Status/Status/Torque reduced
//     Drive/Inputs/In/nState1 @bit 2 <-> STM Status/Status/Warning
//     Drive/Inputs/In/nState2 @bit 3 <-> STM Status/Status/Digital input 1
//     Drive/Inputs/In/nState2 @bit 4 <-> STM Status/Status/Digital input 2
//     Drive/Inputs/In/nState2 @bit 5 <-> STM Status/Status/Sync error
//     Drive/Inputs/In/nState2 @bit 7 <-> STM Status/Status/TxPDO Toggle
//     Drive/Inputs/In/nState4 @bit 1 <-> WcState/InputToggle
//     Drive/Inputs/In/nState4 <-> WcState/WcState
//     Drive/Outputs/Out/nCtrl1 <-> STM Control/Control/Enable
//     Drive/Outputs/Out/nCtrl1 @bit 2 <-> STM Control/Control/Reduce torque
//     Drive/Outputs/Out/nCtrl1 @bit 1 <-> STM Control/Control/Reset
//     Drive/Outputs/Out/nDataOut2[0] <-> STM Velocity/Velocity
//   Axes/SL1K4-SOUTH-M13 <-> Device 1 (EtherCAT)/Power (EK1200)/PLC Junction 1 (EK1122)/X2 TMO FEE EC2 (EK1100)/FEE EC2 E1 (EK1122)/X2 SL1K4-SCATTER/SL1K4-EL5101-E8
//     Enc/Inputs/In/nDataIn1[0] <-> ENC Status compact/Counter value
//     Enc/Inputs/In/nDataIn2[0] <-> ENC Status compact/Latch value
//     Enc/Inputs/In/nState1 @bit 4 <-> ENC Status compact/Status/Counter overflow
//     Enc/Inputs/In/nState1 @bit 3 <-> ENC Status compact/Status/Counter underflow
//     Enc/Inputs/In/nState1 @bit 7 <-> ENC Status compact/Status/Extrapolation stall
//     Enc/Inputs/In/nState1 <-> ENC Status compact/Status/Latch C valid
//     Enc/Inputs/In/nState1 @bit 1 <-> ENC Status compact/Status/Latch extern valid
//     Enc/Inputs/In/nState1 @bit 6 <-> ENC Status compact/Status/Open circuit
//     Enc/Inputs/In/nState1 @bit 2 <-> ENC Status compact/Status/Set counter done
//     Enc/Inputs/In/nState1 @bit 5 <-> ENC Status compact/Status/Status of input status
//     Enc/Inputs/In/nState2 @bit 4 <-> ENC Status compact/Status/Status of extern latch
//     Enc/Inputs/In/nState2 <-> ENC Status compact/Status/Status of input A
//     Enc/Inputs/In/nState2 @bit 1 <-> ENC Status compact/Status/Status of input B
//     Enc/Inputs/In/nState2 @bit 2 <-> ENC Status compact/Status/Status of input C
//     Enc/Inputs/In/nState2 @bit 3 <-> ENC Status compact/Status/Status of input gate
//     Enc/Inputs/In/nState2 @bit 5 <-> ENC Status compact/Status/Sync error
//     Enc/Inputs/In/nState2 @bit 6 <-> ENC Status compact/Status/TxPDO State
//     Enc/Inputs/In/nState2 @bit 7 <-> ENC Status compact/Status/TxPDO Toggle
//     Enc/Inputs/In/nState4 @bit 1 <-> WcState/InputToggle
//     Enc/Inputs/In/nState4 <-> WcState/WcState
//     Enc/Outputs/Out/nCtrl1 <-> ENC Control compact/Control/Enable latch C
//     Enc/Outputs/Out/nCtrl1 @bit 3 <-> ENC Control compact/Control/Enable latch extern on negative edge
//     Enc/Outputs/Out/nCtrl1 @bit 1 <-> ENC Control compact/Control/Enable latch extern on positive edge
//     Enc/Outputs/Out/nCtrl1 @bit 2 <-> ENC Control compact/Control/Set counter
//     Enc/Outputs/Out/nDataOut1[0] <-> ENC Control compact/Set counter value
//   Axes/SL1K4-SOUTH-M13 <-> Device 1 (EtherCAT)/Power (EK1200)/PLC Junction 1 (EK1122)/X2 TMO FEE EC2 (EK1100)/FEE EC2 E1 (EK1122)/X2 SL1K4-SCATTER/SL1K4-EL7031-E7
//     Drive/Inputs/In/nState1 @bit 3 <-> STM Status/Status/Error
//     Drive/Inputs/In/nState1 @bit 5 <-> STM Status/Status/Moving negative
//     Drive/Inputs/In/nState1 @bit 4 <-> STM Status/Status/Moving positive
//     Drive/Inputs/In/nState1 @bit 1 <-> STM Status/Status/Ready
//     Drive/Inputs/In/nState1 <-> STM Status/Status/Ready to enable
//     Drive/Inputs/In/nState1 @bit 6 <-> STM Status/Status/Torque reduced
//     Drive/Inputs/In/nState1 @bit 2 <-> STM Status/Status/Warning
//     Drive/Inputs/In/nState2 @bit 3 <-> STM Status/Status/Digital input 1
//     Drive/Inputs/In/nState2 @bit 4 <-> STM Status/Status/Digital input 2
//     Drive/Inputs/In/nState2 @bit 5 <-> STM Status/Status/Sync error
//     Drive/Inputs/In/nState2 @bit 7 <-> STM Status/Status/TxPDO Toggle
//     Drive/Inputs/In/nState4 @bit 1 <-> WcState/InputToggle
//     Drive/Inputs/In/nState4 <-> WcState/WcState
//     Drive/Outputs/Out/nCtrl1 <-> STM Control/Control/Enable
//     Drive/Outputs/Out/nCtrl1 @bit 2 <-> STM Control/Control/Reduce torque
//     Drive/Outputs/Out/nCtrl1 @bit 1 <-> STM Control/Control/Reset
//     Drive/Outputs/Out/nDataOut2[0] <-> STM Velocity/Velocity
//   Axes/SL1K4-TOP-M11 <-> Device 1 (EtherCAT)/Power (EK1200)/PLC Junction 1 (EK1122)/X2 TMO FEE EC2 (EK1100)/FEE EC2 E1 (EK1122)/X2 SL1K4-SCATTER/SL1K4-EL5101-E4
//     Enc/Inputs/In/nDataIn1[0] <-> ENC Status compact/Counter value
//     Enc/Inputs/In/nDataIn2[0] <-> ENC Status compact/Latch value
//     Enc/Inputs/In/nState1 @bit 4 <-> ENC Status compact/Status/Counter overflow
//     Enc/Inputs/In/nState1 @bit 3 <-> ENC Status compact/Status/Counter underflow
//     Enc/Inputs/In/nState1 @bit 7 <-> ENC Status compact/Status/Extrapolation stall
//     Enc/Inputs/In/nState1 <-> ENC Status compact/Status/Latch C valid
//     Enc/Inputs/In/nState1 @bit 1 <-> ENC Status compact/Status/Latch extern valid
//     Enc/Inputs/In/nState1 @bit 6 <-> ENC Status compact/Status/Open circuit
//     Enc/Inputs/In/nState1 @bit 2 <-> ENC Status compact/Status/Set counter done
//     Enc/Inputs/In/nState1 @bit 5 <-> ENC Status compact/Status/Status of input status
//     Enc/Inputs/In/nState2 @bit 4 <-> ENC Status compact/Status/Status of extern latch
//     Enc/Inputs/In/nState2 <-> ENC Status compact/Status/Status of input A
//     Enc/Inputs/In/nState2 @bit 1 <-> ENC Status compact/Status/Status of input B
//     Enc/Inputs/In/nState2 @bit 2 <-> ENC Status compact/Status/Status of input C
//     Enc/Inputs/In/nState2 @bit 3 <-> ENC Status compact/Status/Status of input gate
//     Enc/Inputs/In/nState2 @bit 5 <-> ENC Status compact/Status/Sync error
//     Enc/Inputs/In/nState2 @bit 6 <-> ENC Status compact/Status/TxPDO State
//     Enc/Inputs/In/nState2 @bit 7 <-> ENC Status compact/Status/TxPDO Toggle
//     Enc/Inputs/In/nState4 @bit 1 <-> WcState/InputToggle
//     Enc/Inputs/In/nState4 <-> WcState/WcState
//     Enc/Outputs/Out/nCtrl1 <-> ENC Control compact/Control/Enable latch C
//     Enc/Outputs/Out/nCtrl1 @bit 3 <-> ENC Control compact/Control/Enable latch extern on negative edge
//     Enc/Outputs/Out/nCtrl1 @bit 1 <-> ENC Control compact/Control/Enable latch extern on positive edge
//     Enc/Outputs/Out/nCtrl1 @bit 2 <-> ENC Control compact/Control/Set counter
//     Enc/Outputs/Out/nDataOut1[0] <-> ENC Control compact/Set counter value
//   Axes/SL1K4-TOP-M11 <-> Device 1 (EtherCAT)/Power (EK1200)/PLC Junction 1 (EK1122)/X2 TMO FEE EC2 (EK1100)/FEE EC2 E1 (EK1122)/X2 SL1K4-SCATTER/SL1K4-EL7031-E3
//     Drive/Inputs/In/nState1 @bit 3 <-> STM Status/Status/Error
//     Drive/Inputs/In/nState1 @bit 5 <-> STM Status/Status/Moving negative
//     Drive/Inputs/In/nState1 @bit 4 <-> STM Status/Status/Moving positive
//     Drive/Inputs/In/nState1 @bit 1 <-> STM Status/Status/Ready
//     Drive/Inputs/In/nState1 <-> STM Status/Status/Ready to enable
//     Drive/Inputs/In/nState1 @bit 6 <-> STM Status/Status/Torque reduced
//     Drive/Inputs/In/nState1 @bit 2 <-> STM Status/Status/Warning
//     Drive/Inputs/In/nState2 @bit 3 <-> STM Status/Status/Digital input 1
//     Drive/Inputs/In/nState2 @bit 4 <-> STM Status/Status/Digital input 2
//     Drive/Inputs/In/nState2 @bit 5 <-> STM Status/Status/Sync error
//     Drive/Inputs/In/nState2 @bit 7 <-> STM Status/Status/TxPDO Toggle
//     Drive/Inputs/In/nState4 @bit 1 <-> WcState/InputToggle
//     Drive/Inputs/In/nState4 <-> WcState/WcState
//     Drive/Outputs/Out/nCtrl1 <-> STM Control/Control/Enable
//     Drive/Outputs/Out/nCtrl1 @bit 2 <-> STM Control/Control/Reduce torque
//     Drive/Outputs/Out/nCtrl1 @bit 1 <-> STM Control/Control/Reset
//     Drive/Outputs/Out/nDataOut2[0] <-> STM Velocity/Velocity
//   (this object) <-> Device 1 (EtherCAT)/Power (EK1200)/PLC Junction 1 (EK1122)/X2 TMO FEE EC2 (EK1100)/FEE EC2 E1 (EK1122)/X1 AL1K4-L2SI (EK1100)/AL1K4-EL5042-E2
//     Enc/Inputs/In/nComState @bit 1 <-> WcState/InputToggle
//     Enc/Inputs/In/nComState <-> WcState/WcState
//     Enc/Inputs/In/nDataIn1 <-> FB Inputs Channel 1/Position
//     Enc/Inputs/In/nState1 @bit 12 <-> FB Inputs Channel 1/Status/Diag
//     Enc/Inputs/In/nState1 @bit 1 <-> FB Inputs Channel 1/Status/Error
//     Enc/Inputs/In/nState1 @bit 14 <-> FB Inputs Channel 1/Status/Input cycle counter
//     Enc/Inputs/In/nState1 @bit 2 <-> FB Inputs Channel 1/Status/Ready
//     Enc/Inputs/In/nState1 @bit 13 <-> FB Inputs Channel 1/Status/TxPDO State
//     Enc/Inputs/In/nState1 <-> FB Inputs Channel 1/Status/Warning
//   (this object) <-> Device 1 (EtherCAT)/Power (EK1200)/PLC Junction 1 (EK1122)/X2 TMO FEE EC2 (EK1100)/FEE EC2 E1 (EK1122)/X1 AL1K4-L2SI (EK1100)/AL1K4-EL7041-E1
//     Drive/Inputs/In/nState1 @bit 3 <-> STM Status/Status/Error
//     Drive/Inputs/In/nState1 @bit 5 <-> STM Status/Status/Moving negative
//     Drive/Inputs/In/nState1 @bit 4 <-> STM Status/Status/Moving positive
//     Drive/Inputs/In/nState1 @bit 1 <-> STM Status/Status/Ready
//     Drive/Inputs/In/nState1 <-> STM Status/Status/Ready to enable
//     Drive/Inputs/In/nState1 @bit 6 <-> STM Status/Status/Torque reduced
//     Drive/Inputs/In/nState1 @bit 2 <-> STM Status/Status/Warning
//     Drive/Inputs/In/nState2 @bit 3 <-> STM Status/Status/Digital input 1
//     Drive/Inputs/In/nState2 @bit 4 <-> STM Status/Status/Digital input 2
//     Drive/Inputs/In/nState2 @bit 5 <-> STM Status/Status/Sync error
//     Drive/Inputs/In/nState2 @bit 7 <-> STM Status/Status/TxPDO Toggle
//     Drive/Inputs/In/nState4 @bit 1 <-> WcState/InputToggle
//     Drive/Inputs/In/nState4 <-> WcState/WcState
//     Drive/Outputs/Out/nCtrl1 <-> STM Control/Control/Enable
//     Drive/Outputs/Out/nCtrl1 @bit 2 <-> STM Control/Control/Reduce torque
//     Drive/Outputs/Out/nCtrl1 @bit 1 <-> STM Control/Control/Reset
//     Drive/Outputs/Out/nDataOut2[0] <-> STM Velocity/Velocity
//   (this object) <-> Device 1 (EtherCAT)/Power (EK1200)/PLC Junction 1 (EK1122)/X1 TMO FEE EC1 (EK1100)/FEE EC1 E1 (EK1122)/X1 IM1K4-XTES (EK1100)/IM1K4-EL7342-E4
//     Drive/Inputs/In/nState1 @bit 3 <-> DCM Status Channel 1/Status/Error
//     Drive/Inputs/In/nState1 @bit 3 <-> DCM Status Channel 2/Status/Error
//     Drive/Inputs/In/nState1 @bit 5 <-> DCM Status Channel 1/Status/Moving negative
//     Drive/Inputs/In/nState1 @bit 5 <-> DCM Status Channel 2/Status/Moving negative
//     Drive/Inputs/In/nState1 @bit 4 <-> DCM Status Channel 1/Status/Moving positive
//     Drive/Inputs/In/nState1 @bit 4 <-> DCM Status Channel 2/Status/Moving positive
//     Drive/Inputs/In/nState1 @bit 1 <-> DCM Status Channel 1/Status/Ready
//     Drive/Inputs/In/nState1 @bit 1 <-> DCM Status Channel 2/Status/Ready
//     Drive/Inputs/In/nState1 <-> DCM Status Channel 1/Status/Ready to enable
//     Drive/Inputs/In/nState1 <-> DCM Status Channel 2/Status/Ready to enable
//     Drive/Inputs/In/nState1 @bit 6 <-> DCM Status Channel 1/Status/Torque reduced
//     Drive/Inputs/In/nState1 @bit 6 <-> DCM Status Channel 2/Status/Torque reduced
//     Drive/Inputs/In/nState1 @bit 2 <-> DCM Status Channel 1/Status/Warning
//     Drive/Inputs/In/nState1 @bit 2 <-> DCM Status Channel 2/Status/Warning
//     Drive/Inputs/In/nState2 @bit 3 <-> DCM Status Channel 1/Status/Digital input 1
//     Drive/Inputs/In/nState2 @bit 4 <-> DCM Status Channel 1/Status/Digital input 2
//     Drive/Inputs/In/nState2 @bit 3 <-> DCM Status Channel 2/Status/Digital input 1
//     Drive/Inputs/In/nState2 @bit 4 <-> DCM Status Channel 2/Status/Digital input 2
//     Drive/Inputs/In/nState2 @bit 5 <-> DCM Status Channel 1/Status/Sync error
//     Drive/Inputs/In/nState2 @bit 5 <-> DCM Status Channel 2/Status/Sync error
//     Drive/Inputs/In/nState2 @bit 7 <-> DCM Status Channel 1/Status/TxPDO Toggle
//     Drive/Inputs/In/nState2 @bit 7 <-> DCM Status Channel 2/Status/TxPDO Toggle
//     Drive/Inputs/In/nState4 @bit 1 <-> WcState/InputToggle
//     Drive/Inputs/In/nState4 <-> WcState/WcState
//     Drive/Outputs/Out/nCtrl1 <-> DCM Control Channel 1/Control/Enable
//     Drive/Outputs/Out/nCtrl1 <-> DCM Control Channel 2/Control/Enable
//     Drive/Outputs/Out/nCtrl1 @bit 2 <-> DCM Control Channel 1/Control/Reduce torque
//     Drive/Outputs/Out/nCtrl1 @bit 2 <-> DCM Control Channel 2/Control/Reduce torque
//     Drive/Outputs/Out/nCtrl1 @bit 1 <-> DCM Control Channel 1/Control/Reset
//     Drive/Outputs/Out/nCtrl1 @bit 1 <-> DCM Control Channel 2/Control/Reset
//     Drive/Outputs/Out/nDataOut2[0] <-> DCM Velocity Channel 1/Velocity
//     Drive/Outputs/Out/nDataOut2[0] <-> DCM Velocity Channel 2/Velocity
//     Enc/Inputs/In/nDataIn1[0] <-> ENC Status compact Channel 1/Counter value
//     Enc/Inputs/In/nDataIn1[0] <-> ENC Status compact Channel 2/Counter value
//     Enc/Inputs/In/nDataIn2[0] <-> ENC Status compact Channel 1/Latch value
//     Enc/Inputs/In/nDataIn2[0] <-> ENC Status compact Channel 2/Latch value
//     Enc/Inputs/In/nState1 @bit 4 <-> ENC Status compact Channel 1/Status/Counter overflow
//     Enc/Inputs/In/nState1 @bit 4 <-> ENC Status compact Channel 2/Status/Counter overflow
//     Enc/Inputs/In/nState1 @bit 3 <-> ENC Status compact Channel 1/Status/Counter underflow
//     Enc/Inputs/In/nState1 @bit 3 <-> ENC Status compact Channel 2/Status/Counter underflow
//     Enc/Inputs/In/nState1 @bit 7 <-> ENC Status compact Channel 1/Status/Extrapolation stall
//     Enc/Inputs/In/nState1 @bit 7 <-> ENC Status compact Channel 2/Status/Extrapolation stall
//     Enc/Inputs/In/nState1 @bit 1 <-> ENC Status compact Channel 1/Status/Latch extern valid
//     Enc/Inputs/In/nState1 @bit 1 <-> ENC Status compact Channel 2/Status/Latch extern valid
//     Enc/Inputs/In/nState1 @bit 2 <-> ENC Status compact Channel 1/Status/Set counter done
//     Enc/Inputs/In/nState1 @bit 2 <-> ENC Status compact Channel 2/Status/Set counter done
//     Enc/Inputs/In/nState2 @bit 4 <-> ENC Status compact Channel 1/Status/Status of extern latch
//     Enc/Inputs/In/nState2 @bit 4 <-> ENC Status compact Channel 2/Status/Status of extern latch
//     Enc/Inputs/In/nState2 <-> ENC Status compact Channel 1/Status/Status of input A
//     Enc/Inputs/In/nState2 <-> ENC Status compact Channel 2/Status/Status of input A
//     Enc/Inputs/In/nState2 @bit 1 <-> ENC Status compact Channel 1/Status/Status of input B
//     Enc/Inputs/In/nState2 @bit 1 <-> ENC Status compact Channel 2/Status/Status of input B
//     Enc/Inputs/In/nState2 @bit 5 <-> ENC Status compact Channel 1/Status/Sync error
//     Enc/Inputs/In/nState2 @bit 5 <-> ENC Status compact Channel 2/Status/Sync error
//     Enc/Inputs/In/nState2 @bit 7 <-> ENC Status compact Channel 1/Status/TxPDO Toggle
//     Enc/Inputs/In/nState2 @bit 7 <-> ENC Status compact Channel 2/Status/TxPDO Toggle
//     Enc/Inputs/In/nState4 @bit 1 <-> WcState/InputToggle
//     Enc/Inputs/In/nState4 <-> WcState/WcState
//     Enc/Outputs/Out/nCtrl1 @bit 3 <-> ENC Control compact Channel 1/Control/Enable latch extern on negative edge
//     Enc/Outputs/Out/nCtrl1 @bit 3 <-> ENC Control compact Channel 2/Control/Enable latch extern on negative edge
//     Enc/Outputs/Out/nCtrl1 @bit 1 <-> ENC Control compact Channel 1/Control/Enable latch extern on positive edge
//     Enc/Outputs/Out/nCtrl1 @bit 1 <-> ENC Control compact Channel 2/Control/Enable latch extern on positive edge
//     Enc/Outputs/Out/nCtrl1 @bit 2 <-> ENC Control compact Channel 1/Control/Set counter
//     Enc/Outputs/Out/nCtrl1 @bit 2 <-> ENC Control compact Channel 2/Control/Set counter
//     Enc/Outputs/Out/nDataOut1[0] <-> ENC Control compact Channel 1/Set counter value
//     Enc/Outputs/Out/nDataOut1[0] <-> ENC Control compact Channel 2/Set counter value
//   (this object) <-> Device 1 (EtherCAT)/Power (EK1200)/PLC Junction 1 (EK1122)/X2 TMO FEE EC2 (EK1100)/FEE EC2 E2 (EK1122)/X1 IM2K4-PPM (EK1100)/IM2K4-EL5042-E2
//     Enc/Inputs/In/nComState @bit 1 <-> WcState/InputToggle
//     Enc/Inputs/In/nComState <-> WcState/WcState
//     Enc/Inputs/In/nDataIn1 <-> FB Inputs Channel 1/Position
//     Enc/Inputs/In/nState1 @bit 12 <-> FB Inputs Channel 1/Status/Diag
//     Enc/Inputs/In/nState1 @bit 1 <-> FB Inputs Channel 1/Status/Error
//     Enc/Inputs/In/nState1 @bit 14 <-> FB Inputs Channel 1/Status/Input cycle counter
//     Enc/Inputs/In/nState1 @bit 2 <-> FB Inputs Channel 1/Status/Ready
//     Enc/Inputs/In/nState1 @bit 13 <-> FB Inputs Channel 1/Status/TxPDO State
//     Enc/Inputs/In/nState1 <-> FB Inputs Channel 1/Status/Warning
//   (this object) <-> Device 1 (EtherCAT)/Power (EK1200)/PLC Junction 1 (EK1122)/X2 TMO FEE EC2 (EK1100)/FEE EC2 E2 (EK1122)/X1 IM2K4-PPM (EK1100)/IM2K4-EL7041-E1
//     Drive/Inputs/In/nState1 @bit 3 <-> STM Status/Status/Error
//     Drive/Inputs/In/nState1 @bit 5 <-> STM Status/Status/Moving negative
//     Drive/Inputs/In/nState1 @bit 4 <-> STM Status/Status/Moving positive
//     Drive/Inputs/In/nState1 @bit 1 <-> STM Status/Status/Ready
//     Drive/Inputs/In/nState1 <-> STM Status/Status/Ready to enable
//     Drive/Inputs/In/nState1 @bit 6 <-> STM Status/Status/Torque reduced
//     Drive/Inputs/In/nState1 @bit 2 <-> STM Status/Status/Warning
//     Drive/Inputs/In/nState2 @bit 3 <-> STM Status/Status/Digital input 1
//     Drive/Inputs/In/nState2 @bit 4 <-> STM Status/Status/Digital input 2
//     Drive/Inputs/In/nState2 @bit 5 <-> STM Status/Status/Sync error
//     Drive/Inputs/In/nState2 @bit 7 <-> STM Status/Status/TxPDO Toggle
//     Drive/Inputs/In/nState4 @bit 1 <-> WcState/InputToggle
//     Drive/Inputs/In/nState4 <-> WcState/WcState
//     Drive/Outputs/Out/nCtrl1 <-> STM Control/Control/Enable
//     Drive/Outputs/Out/nCtrl1 @bit 2 <-> STM Control/Control/Reduce torque
//     Drive/Outputs/Out/nCtrl1 @bit 1 <-> STM Control/Control/Reset
//     Drive/Outputs/Out/nDataOut2[0] <-> STM Velocity/Velocity
//   (this object) <-> Device 1 (EtherCAT)/Power (EK1200)/PLC Junction 1 (EK1122)/X1 TMO FEE EC1 (EK1100)/FEE EC1 E1 (EK1122)/X2-ST1K4-TEST (EK1100)/ST1K4-EL7041-E4
//     Drive/Inputs/In/nState1 @bit 3 <-> STM Status/Status/Error
//     Drive/Inputs/In/nState1 @bit 5 <-> STM Status/Status/Moving negative
//     Drive/Inputs/In/nState1 @bit 4 <-> STM Status/Status/Moving positive
//     Drive/Inputs/In/nState1 @bit 1 <-> STM Status/Status/Ready
//     Drive/Inputs/In/nState1 <-> STM Status/Status/Ready to enable
//     Drive/Inputs/In/nState1 @bit 6 <-> STM Status/Status/Torque reduced
//     Drive/Inputs/In/nState1 @bit 2 <-> STM Status/Status/Warning
//     Drive/Inputs/In/nState2 @bit 3 <-> STM Status/Status/Digital input 1
//     Drive/Inputs/In/nState2 @bit 4 <-> STM Status/Status/Digital input 2
//     Drive/Inputs/In/nState2 @bit 5 <-> STM Status/Status/Sync error
//     Drive/Inputs/In/nState2 @bit 7 <-> STM Status/Status/TxPDO Toggle
//     Drive/Inputs/In/nState4 @bit 1 <-> WcState/InputToggle
//     Drive/Inputs/In/nState4 <-> WcState/WcState
//     Drive/Outputs/Out/nCtrl1 <-> STM Control/Control/Enable
//     Drive/Outputs/Out/nCtrl1 @bit 2 <-> STM Control/Control/Reduce torque
//     Drive/Outputs/Out/nCtrl1 @bit 1 <-> STM Control/Control/Reset
//     Drive/Outputs/Out/nDataOut2[0] <-> STM Velocity/Velocity
//     Enc/Inputs/In/nDataIn1[0] <-> ENC Status compact/Counter value
//     Enc/Inputs/In/nDataIn2[0] <-> ENC Status compact/Latch value
//     Enc/Inputs/In/nState1 @bit 4 <-> ENC Status compact/Status/Counter overflow
//     Enc/Inputs/In/nState1 @bit 3 <-> ENC Status compact/Status/Counter underflow
//     Enc/Inputs/In/nState1 @bit 7 <-> ENC Status compact/Status/Extrapolation stall
//     Enc/Inputs/In/nState1 <-> ENC Status compact/Status/Latch C valid
//     Enc/Inputs/In/nState1 @bit 1 <-> ENC Status compact/Status/Latch extern valid
//     Enc/Inputs/In/nState1 @bit 2 <-> ENC Status compact/Status/Set counter done
//     Enc/Inputs/In/nState2 @bit 4 <-> ENC Status compact/Status/Status of extern latch
//     Enc/Inputs/In/nState2 <-> ENC Status compact/Status/Status of input A
//     Enc/Inputs/In/nState2 @bit 1 <-> ENC Status compact/Status/Status of input B
//     Enc/Inputs/In/nState2 @bit 2 <-> ENC Status compact/Status/Status of input C
//     Enc/Inputs/In/nState2 @bit 5 <-> ENC Status compact/Status/Sync error
//     Enc/Inputs/In/nState2 @bit 7 <-> ENC Status compact/Status/TxPDO Toggle
//     Enc/Inputs/In/nState4 @bit 1 <-> WcState/InputToggle
//     Enc/Inputs/In/nState4 <-> WcState/WcState
//     Enc/Outputs/Out/nCtrl1 <-> ENC Control compact/Control/Enable latch C
//     Enc/Outputs/Out/nCtrl1 @bit 3 <-> ENC Control compact/Control/Enable latch extern on negative edge
//     Enc/Outputs/Out/nCtrl1 @bit 1 <-> ENC Control compact/Control/Enable latch extern on positive edge
//     Enc/Outputs/Out/nCtrl1 @bit 2 <-> ENC Control compact/Control/Set counter
//     Enc/Outputs/Out/nDataOut1[0] <-> ENC Control compact/Set counter value
//   (this object) <-> Device 1 (EtherCAT)/Power (EK1200)/PLC Junction 2 (EK1122)/PLC Coupler 1(EK1100)/PLC Junction 5 (EK1122)/IM3K4-PPM (EK1100)/IM3K4-EL5042-E2
//     Enc/Inputs/In/nComState @bit 1 <-> WcState/InputToggle
//     Enc/Inputs/In/nComState <-> WcState/WcState
//     Enc/Inputs/In/nDataIn1 <-> FB Inputs Channel 1/Position
//     Enc/Inputs/In/nState1 @bit 12 <-> FB Inputs Channel 1/Status/Diag
//     Enc/Inputs/In/nState1 @bit 1 <-> FB Inputs Channel 1/Status/Error
//     Enc/Inputs/In/nState1 @bit 14 <-> FB Inputs Channel 1/Status/Input cycle counter
//     Enc/Inputs/In/nState1 @bit 2 <-> FB Inputs Channel 1/Status/Ready
//     Enc/Inputs/In/nState1 @bit 13 <-> FB Inputs Channel 1/Status/TxPDO State
//     Enc/Inputs/In/nState1 <-> FB Inputs Channel 1/Status/Warning
//   (this object) <-> Device 1 (EtherCAT)/Power (EK1200)/PLC Junction 2 (EK1122)/PLC Coupler 1(EK1100)/PLC Junction 5 (EK1122)/IM3K4-PPM (EK1100)/IM3K4-EL7041-E1
//     Drive/Inputs/In/nState1 @bit 3 <-> STM Status/Status/Error
//     Drive/Inputs/In/nState1 @bit 5 <-> STM Status/Status/Moving negative
//     Drive/Inputs/In/nState1 @bit 4 <-> STM Status/Status/Moving positive
//     Drive/Inputs/In/nState1 @bit 1 <-> STM Status/Status/Ready
//     Drive/Inputs/In/nState1 <-> STM Status/Status/Ready to enable
//     Drive/Inputs/In/nState1 @bit 6 <-> STM Status/Status/Torque reduced
//     Drive/Inputs/In/nState1 @bit 2 <-> STM Status/Status/Warning
//     Drive/Inputs/In/nState2 @bit 5 <-> STM Status/Status/Sync error
//     Drive/Inputs/In/nState2 @bit 7 <-> STM Status/Status/TxPDO Toggle
//     Drive/Inputs/In/nState4 @bit 1 <-> WcState/InputToggle
//     Drive/Inputs/In/nState4 <-> WcState/WcState
//     Drive/Outputs/Out/nCtrl1 <-> STM Control/Control/Enable
//     Drive/Outputs/Out/nCtrl1 @bit 2 <-> STM Control/Control/Reduce torque
//     Drive/Outputs/Out/nCtrl1 @bit 1 <-> STM Control/Control/Reset
//     Drive/Outputs/Out/nDataOut2[0] <-> STM Velocity/Velocity
//   (this object) <-> Device 1 (EtherCAT)/Power (EK1200)/PLC Junction 2 (EK1122)/PLC Coupler 1(EK1100)/PLC Junction 5 (EK1122)/IM4K4-PPM (EK1100)/IM4K4-EL5042-E2
//     Enc/Inputs/In/nComState @bit 1 <-> WcState/InputToggle
//     Enc/Inputs/In/nComState <-> WcState/WcState
//     Enc/Inputs/In/nDataIn1 <-> FB Inputs Channel 1/Position
//     Enc/Inputs/In/nState1 @bit 12 <-> FB Inputs Channel 1/Status/Diag
//     Enc/Inputs/In/nState1 @bit 1 <-> FB Inputs Channel 1/Status/Error
//     Enc/Inputs/In/nState1 @bit 14 <-> FB Inputs Channel 1/Status/Input cycle counter
//     Enc/Inputs/In/nState1 @bit 2 <-> FB Inputs Channel 1/Status/Ready
//     Enc/Inputs/In/nState1 @bit 13 <-> FB Inputs Channel 1/Status/TxPDO State
//     Enc/Inputs/In/nState1 <-> FB Inputs Channel 1/Status/Warning
//   (this object) <-> Device 1 (EtherCAT)/Power (EK1200)/PLC Junction 2 (EK1122)/PLC Coupler 1(EK1100)/PLC Junction 5 (EK1122)/IM4K4-PPM (EK1100)/IM4K4-EL7041-E1
//     Drive/Inputs/In/nState1 @bit 3 <-> STM Status/Status/Error
//     Drive/Inputs/In/nState1 @bit 5 <-> STM Status/Status/Moving negative
//     Drive/Inputs/In/nState1 @bit 4 <-> STM Status/Status/Moving positive
//     Drive/Inputs/In/nState1 @bit 1 <-> STM Status/Status/Ready
//     Drive/Inputs/In/nState1 <-> STM Status/Status/Ready to enable
//     Drive/Inputs/In/nState1 @bit 6 <-> STM Status/Status/Torque reduced
//     Drive/Inputs/In/nState1 @bit 2 <-> STM Status/Status/Warning
//     Drive/Inputs/In/nState2 @bit 3 <-> STM Status/Status/Digital input 1
//     Drive/Inputs/In/nState2 @bit 4 <-> STM Status/Status/Digital input 2
//     Drive/Inputs/In/nState2 @bit 5 <-> STM Status/Status/Sync error
//     Drive/Inputs/In/nState2 @bit 7 <-> STM Status/Status/TxPDO Toggle
//     Drive/Inputs/In/nState4 @bit 1 <-> WcState/InputToggle
//     Drive/Inputs/In/nState4 <-> WcState/WcState
//     Drive/Outputs/Out/nCtrl1 <-> STM Control/Control/Enable
//     Drive/Outputs/Out/nCtrl1 @bit 2 <-> STM Control/Control/Reduce torque
//     Drive/Outputs/Out/nCtrl1 @bit 1 <-> STM Control/Control/Reset
//     Drive/Outputs/Out/nDataOut2[0] <-> STM Velocity/Velocity
//   (this object) <-> Device 1 (EtherCAT)/Power (EK1200)/PLC Junction 2 (EK1122)/PLC Coupler 2 (EK1100)/PLC Junction 8 (EK1122)/IM5K4-PPM (EK1100)/IM5K4-EL5042-E2
//     Enc/Inputs/In/nComState @bit 1 <-> WcState/InputToggle
//     Enc/Inputs/In/nComState <-> WcState/WcState
//     Enc/Inputs/In/nDataIn1 <-> FB Inputs Channel 1/Position
//     Enc/Inputs/In/nState1 @bit 12 <-> FB Inputs Channel 1/Status/Diag
//     Enc/Inputs/In/nState1 @bit 1 <-> FB Inputs Channel 1/Status/Error
//     Enc/Inputs/In/nState1 @bit 14 <-> FB Inputs Channel 1/Status/Input cycle counter
//     Enc/Inputs/In/nState1 @bit 2 <-> FB Inputs Channel 1/Status/Ready
//     Enc/Inputs/In/nState1 @bit 13 <-> FB Inputs Channel 1/Status/TxPDO State
//     Enc/Inputs/In/nState1 <-> FB Inputs Channel 1/Status/Warning
//   (this object) <-> Device 1 (EtherCAT)/Power (EK1200)/PLC Junction 2 (EK1122)/PLC Coupler 2 (EK1100)/PLC Junction 8 (EK1122)/IM5K4-PPM (EK1100)/IM5K4-EL7041-E1
//     Drive/Inputs/In/nState1 @bit 3 <-> STM Status/Status/Error
//     Drive/Inputs/In/nState1 @bit 5 <-> STM Status/Status/Moving negative
//     Drive/Inputs/In/nState1 @bit 4 <-> STM Status/Status/Moving positive
//     Drive/Inputs/In/nState1 @bit 1 <-> STM Status/Status/Ready
//     Drive/Inputs/In/nState1 <-> STM Status/Status/Ready to enable
//     Drive/Inputs/In/nState1 @bit 6 <-> STM Status/Status/Torque reduced
//     Drive/Inputs/In/nState1 @bit 2 <-> STM Status/Status/Warning
//     Drive/Inputs/In/nState2 @bit 3 <-> STM Status/Status/Digital input 1
//     Drive/Inputs/In/nState2 @bit 4 <-> STM Status/Status/Digital input 2
//     Drive/Inputs/In/nState2 @bit 5 <-> STM Status/Status/Sync error
//     Drive/Inputs/In/nState2 @bit 7 <-> STM Status/Status/TxPDO Toggle
//     Drive/Inputs/In/nState4 @bit 1 <-> WcState/InputToggle
//     Drive/Inputs/In/nState4 <-> WcState/WcState
//     Drive/Outputs/Out/nCtrl1 <-> STM Control/Control/Enable
//     Drive/Outputs/Out/nCtrl1 @bit 2 <-> STM Control/Control/Reduce torque
//     Drive/Outputs/Out/nCtrl1 @bit 1 <-> STM Control/Control/Reset
//     Drive/Outputs/Out/nDataOut2[0] <-> STM Velocity/Velocity
//   (this object) <-> Device 1 (EtherCAT)/Power (EK1200)/PLC Junction 2 (EK1122)/PLC Coupler 2 (EK1100)/PLC Junction 10 (EK1122)/PF1K4-WFS (EK1100)/PF1K4-EL5042-E3
//     Enc/Inputs/In/nComState @bit 1 <-> WcState/InputToggle
//     Enc/Inputs/In/nComState <-> WcState/WcState
//     Enc/Inputs/In/nDataIn1 <-> FB Inputs Channel 2/Position
//     Enc/Inputs/In/nState1 @bit 12 <-> FB Inputs Channel 2/Status/Diag
//     Enc/Inputs/In/nState1 @bit 1 <-> FB Inputs Channel 2/Status/Error
//     Enc/Inputs/In/nState1 @bit 14 <-> FB Inputs Channel 2/Status/Input cycle counter
//     Enc/Inputs/In/nState1 @bit 2 <-> FB Inputs Channel 2/Status/Ready
//     Enc/Inputs/In/nState1 @bit 13 <-> FB Inputs Channel 2/Status/TxPDO State
//     Enc/Inputs/In/nState1 <-> FB Inputs Channel 2/Status/Warning
//   (this object) <-> Device 1 (EtherCAT)/Power (EK1200)/PLC Junction 2 (EK1122)/PLC Coupler 2 (EK1100)/PLC Junction 10 (EK1122)/PF1K4-WFS (EK1100)/PF1K4-EL7041-E1
//     Drive/Inputs/In/nState1 @bit 3 <-> STM Status/Status/Error
//     Drive/Inputs/In/nState1 @bit 5 <-> STM Status/Status/Moving negative
//     Drive/Inputs/In/nState1 @bit 4 <-> STM Status/Status/Moving positive
//     Drive/Inputs/In/nState1 @bit 1 <-> STM Status/Status/Ready
//     Drive/Inputs/In/nState1 <-> STM Status/Status/Ready to enable
//     Drive/Inputs/In/nState1 @bit 6 <-> STM Status/Status/Torque reduced
//     Drive/Inputs/In/nState1 @bit 2 <-> STM Status/Status/Warning
//     Drive/Inputs/In/nState2 @bit 3 <-> STM Status/Status/Digital input 1
//     Drive/Inputs/In/nState2 @bit 4 <-> STM Status/Status/Digital input 2
//     Drive/Inputs/In/nState2 @bit 5 <-> STM Status/Status/Sync error
//     Drive/Inputs/In/nState2 @bit 7 <-> STM Status/Status/TxPDO Toggle
//     Drive/Inputs/In/nState4 @bit 1 <-> WcState/InputToggle
//     Drive/Inputs/In/nState4 <-> WcState/WcState
//     Drive/Outputs/Out/nCtrl1 <-> STM Control/Control/Enable
//     Drive/Outputs/Out/nCtrl1 @bit 2 <-> STM Control/Control/Reduce torque
//     Drive/Outputs/Out/nCtrl1 @bit 1 <-> STM Control/Control/Reset
//     Drive/Outputs/Out/nDataOut2[0] <-> STM Velocity/Velocity
//   (this object) <-> Device 1 (EtherCAT)/Power (EK1200)/PLC Junction 2 (EK1122)/PLC Coupler 2 (EK1100)/PLC Junction 10 (EK1122)/PF1K4-WFS (EK1100)/PF1K4-EL7041-E2
//     Drive/Inputs/In/nState1 @bit 3 <-> STM Status/Status/Error
//     Drive/Inputs/In/nState1 @bit 5 <-> STM Status/Status/Moving negative
//     Drive/Inputs/In/nState1 @bit 4 <-> STM Status/Status/Moving positive
//     Drive/Inputs/In/nState1 @bit 1 <-> STM Status/Status/Ready
//     Drive/Inputs/In/nState1 <-> STM Status/Status/Ready to enable
//     Drive/Inputs/In/nState1 @bit 6 <-> STM Status/Status/Torque reduced
//     Drive/Inputs/In/nState1 @bit 2 <-> STM Status/Status/Warning
//     Drive/Inputs/In/nState2 @bit 3 <-> STM Status/Status/Digital input 1
//     Drive/Inputs/In/nState2 @bit 4 <-> STM Status/Status/Digital input 2
//     Drive/Inputs/In/nState2 @bit 5 <-> STM Status/Status/Sync error
//     Drive/Inputs/In/nState2 @bit 7 <-> STM Status/Status/TxPDO Toggle
//     Drive/Inputs/In/nState4 @bit 1 <-> WcState/InputToggle
//     Drive/Inputs/In/nState4 <-> WcState/WcState
//     Drive/Outputs/Out/nCtrl1 <-> STM Control/Control/Enable
//     Drive/Outputs/Out/nCtrl1 @bit 2 <-> STM Control/Control/Reduce torque
//     Drive/Outputs/Out/nCtrl1 @bit 1 <-> STM Control/Control/Reset
//     Drive/Outputs/Out/nDataOut2[0] <-> STM Velocity/Velocity
//   (this object) <-> Device 1 (EtherCAT)/Power (EK1200)/PLC Junction 2 (EK1122)/PLC Coupler 1(EK1100)/PLC Junction 6 (EK1122)/LI1K4-LIC (EK1100)/LI1K4-EL5042-E2
//     Enc/Inputs/In/nComState @bit 1 <-> WcState/InputToggle
//     Enc/Inputs/In/nComState <-> WcState/WcState
//     Enc/Inputs/In/nDataIn1 <-> FB Inputs Channel 1/Position
//     Enc/Inputs/In/nState1 @bit 12 <-> FB Inputs Channel 1/Status/Diag
//     Enc/Inputs/In/nState1 @bit 1 <-> FB Inputs Channel 1/Status/Error
//     Enc/Inputs/In/nState1 @bit 14 <-> FB Inputs Channel 1/Status/Input cycle counter
//     Enc/Inputs/In/nState1 @bit 2 <-> FB Inputs Channel 1/Status/Ready
//     Enc/Inputs/In/nState1 @bit 13 <-> FB Inputs Channel 1/Status/TxPDO State
//     Enc/Inputs/In/nState1 <-> FB Inputs Channel 1/Status/Warning
//   (this object) <-> Device 1 (EtherCAT)/Power (EK1200)/PLC Junction 2 (EK1122)/PLC Coupler 1(EK1100)/PLC Junction 6 (EK1122)/LI1K4-LIC (EK1100)/LI1K4-EL7041-E1
//     Drive/Inputs/In/nState1 @bit 3 <-> STM Status/Status/Error
//     Drive/Inputs/In/nState1 @bit 5 <-> STM Status/Status/Moving negative
//     Drive/Inputs/In/nState1 @bit 4 <-> STM Status/Status/Moving positive
//     Drive/Inputs/In/nState1 @bit 1 <-> STM Status/Status/Ready
//     Drive/Inputs/In/nState1 <-> STM Status/Status/Ready to enable
//     Drive/Inputs/In/nState1 @bit 6 <-> STM Status/Status/Torque reduced
//     Drive/Inputs/In/nState1 @bit 2 <-> STM Status/Status/Warning
//     Drive/Inputs/In/nState2 @bit 3 <-> STM Status/Status/Digital input 1
//     Drive/Inputs/In/nState2 @bit 4 <-> STM Status/Status/Digital input 2
//     Drive/Inputs/In/nState2 @bit 5 <-> STM Status/Status/Sync error
//     Drive/Inputs/In/nState2 @bit 7 <-> STM Status/Status/TxPDO Toggle
//     Drive/Inputs/In/nState4 @bit 1 <-> WcState/InputToggle
//     Drive/Inputs/In/nState4 <-> WcState/WcState
//     Drive/Outputs/Out/nCtrl1 <-> STM Control/Control/Enable
//     Drive/Outputs/Out/nCtrl1 @bit 2 <-> STM Control/Control/Reduce torque
//     Drive/Outputs/Out/nCtrl1 @bit 1 <-> STM Control/Control/Reset
//     Drive/Outputs/Out/nDataOut2[0] <-> STM Velocity/Velocity
//   (this object) <-> Device 1 (EtherCAT)/Power (EK1200)/PLC Junction 2 (EK1122)/PLC Coupler 2 (EK1100)/PLC Junction 7 (EK1122)/TM1K4-ATM (EK1100)/TM1K4-EL5042-E3
//     Enc/Inputs/In/nComState @bit 1 <-> WcState/InputToggle
//     Enc/Inputs/In/nComState <-> WcState/WcState
//     Enc/Inputs/In/nDataIn1 <-> FB Inputs Channel 1/Position
//     Enc/Inputs/In/nDataIn1 <-> FB Inputs Channel 2/Position
//     Enc/Inputs/In/nState1 @bit 12 <-> FB Inputs Channel 1/Status/Diag
//     Enc/Inputs/In/nState1 @bit 12 <-> FB Inputs Channel 2/Status/Diag
//     Enc/Inputs/In/nState1 @bit 1 <-> FB Inputs Channel 1/Status/Error
//     Enc/Inputs/In/nState1 @bit 1 <-> FB Inputs Channel 2/Status/Error
//     Enc/Inputs/In/nState1 @bit 14 <-> FB Inputs Channel 1/Status/Input cycle counter
//     Enc/Inputs/In/nState1 @bit 14 <-> FB Inputs Channel 2/Status/Input cycle counter
//     Enc/Inputs/In/nState1 @bit 2 <-> FB Inputs Channel 1/Status/Ready
//     Enc/Inputs/In/nState1 @bit 2 <-> FB Inputs Channel 2/Status/Ready
//     Enc/Inputs/In/nState1 @bit 13 <-> FB Inputs Channel 1/Status/TxPDO State
//     Enc/Inputs/In/nState1 @bit 13 <-> FB Inputs Channel 2/Status/TxPDO State
//     Enc/Inputs/In/nState1 <-> FB Inputs Channel 1/Status/Warning
//     Enc/Inputs/In/nState1 <-> FB Inputs Channel 2/Status/Warning
//   (this object) <-> Device 1 (EtherCAT)/Power (EK1200)/PLC Junction 2 (EK1122)/PLC Coupler 2 (EK1100)/PLC Junction 7 (EK1122)/TM1K4-ATM (EK1100)/TM1K4-EL7041-E1
//     Drive/Inputs/In/nState1 @bit 3 <-> STM Status/Status/Error
//     Drive/Inputs/In/nState1 @bit 5 <-> STM Status/Status/Moving negative
//     Drive/Inputs/In/nState1 @bit 4 <-> STM Status/Status/Moving positive
//     Drive/Inputs/In/nState1 @bit 1 <-> STM Status/Status/Ready
//     Drive/Inputs/In/nState1 <-> STM Status/Status/Ready to enable
//     Drive/Inputs/In/nState1 @bit 6 <-> STM Status/Status/Torque reduced
//     Drive/Inputs/In/nState1 @bit 2 <-> STM Status/Status/Warning
//     Drive/Inputs/In/nState2 @bit 3 <-> STM Status/Status/Digital input 1
//     Drive/Inputs/In/nState2 @bit 4 <-> STM Status/Status/Digital input 2
//     Drive/Inputs/In/nState2 @bit 5 <-> STM Status/Status/Sync error
//     Drive/Inputs/In/nState2 @bit 7 <-> STM Status/Status/TxPDO Toggle
//     Drive/Inputs/In/nState4 @bit 1 <-> WcState/InputToggle
//     Drive/Inputs/In/nState4 <-> WcState/WcState
//     Drive/Outputs/Out/nCtrl1 <-> STM Control/Control/Enable
//     Drive/Outputs/Out/nCtrl1 @bit 2 <-> STM Control/Control/Reduce torque
//     Drive/Outputs/Out/nCtrl1 @bit 1 <-> STM Control/Control/Reset
//     Drive/Outputs/Out/nDataOut2[0] <-> STM Velocity/Velocity
//   (this object) <-> Device 1 (EtherCAT)/Power (EK1200)/PLC Junction 2 (EK1122)/PLC Coupler 2 (EK1100)/PLC Junction 7 (EK1122)/TM1K4-ATM (EK1100)/TM1K4-EL7041-E2
//     Drive/Inputs/In/nState1 @bit 3 <-> STM Status/Status/Error
//     Drive/Inputs/In/nState1 @bit 5 <-> STM Status/Status/Moving negative
//     Drive/Inputs/In/nState1 @bit 4 <-> STM Status/Status/Moving positive
//     Drive/Inputs/In/nState1 @bit 1 <-> STM Status/Status/Ready
//     Drive/Inputs/In/nState1 <-> STM Status/Status/Ready to enable
//     Drive/Inputs/In/nState1 @bit 6 <-> STM Status/Status/Torque reduced
//     Drive/Inputs/In/nState1 @bit 2 <-> STM Status/Status/Warning
//     Drive/Inputs/In/nState2 @bit 3 <-> STM Status/Status/Digital input 1
//     Drive/Inputs/In/nState2 @bit 4 <-> STM Status/Status/Digital input 2
//     Drive/Inputs/In/nState2 @bit 5 <-> STM Status/Status/Sync error
//     Drive/Inputs/In/nState2 @bit 7 <-> STM Status/Status/TxPDO Toggle
//     Drive/Inputs/In/nState4 @bit 1 <-> WcState/InputToggle
//     Drive/Inputs/In/nState4 <-> WcState/WcState
//     Drive/Outputs/Out/nCtrl1 <-> STM Control/Control/Enable
//     Drive/Outputs/Out/nCtrl1 @bit 2 <-> STM Control/Control/Reduce torque
//     Drive/Outputs/Out/nCtrl1 @bit 1 <-> STM Control/Control/Reset
//     Drive/Outputs/Out/nDataOut2[0] <-> STM Velocity/Velocity
//   (this object) <-> Device 1 (EtherCAT)/Power (EK1200)/PLC Junction 2 (EK1122)/PLC Coupler 2 (EK1100)/PLC Junction 9 (EK1122)/X2 SL2K4-SCATTER/SL2K4-EL5101-E2
//     Enc/Inputs/In/nDataIn1[0] <-> ENC Status compact/Counter value
//     Enc/Inputs/In/nDataIn2[0] <-> ENC Status compact/Latch value
//     Enc/Inputs/In/nState1 @bit 4 <-> ENC Status compact/Status/Counter overflow
//     Enc/Inputs/In/nState1 @bit 3 <-> ENC Status compact/Status/Counter underflow
//     Enc/Inputs/In/nState1 @bit 7 <-> ENC Status compact/Status/Extrapolation stall
//     Enc/Inputs/In/nState1 <-> ENC Status compact/Status/Latch C valid
//     Enc/Inputs/In/nState1 @bit 1 <-> ENC Status compact/Status/Latch extern valid
//     Enc/Inputs/In/nState1 @bit 6 <-> ENC Status compact/Status/Open circuit
//     Enc/Inputs/In/nState1 @bit 2 <-> ENC Status compact/Status/Set counter done
//     Enc/Inputs/In/nState1 @bit 5 <-> ENC Status compact/Status/Status of input status
//     Enc/Inputs/In/nState2 @bit 4 <-> ENC Status compact/Status/Status of extern latch
//     Enc/Inputs/In/nState2 <-> ENC Status compact/Status/Status of input A
//     Enc/Inputs/In/nState2 @bit 1 <-> ENC Status compact/Status/Status of input B
//     Enc/Inputs/In/nState2 @bit 2 <-> ENC Status compact/Status/Status of input C
//     Enc/Inputs/In/nState2 @bit 3 <-> ENC Status compact/Status/Status of input gate
//     Enc/Inputs/In/nState2 @bit 5 <-> ENC Status compact/Status/Sync error
//     Enc/Inputs/In/nState2 @bit 6 <-> ENC Status compact/Status/TxPDO State
//     Enc/Inputs/In/nState2 @bit 7 <-> ENC Status compact/Status/TxPDO Toggle
//     Enc/Inputs/In/nState4 @bit 1 <-> WcState/InputToggle
//     Enc/Inputs/In/nState4 <-> WcState/WcState
//     Enc/Outputs/Out/nCtrl1 <-> ENC Control compact/Control/Enable latch C
//     Enc/Outputs/Out/nCtrl1 @bit 3 <-> ENC Control compact/Control/Enable latch extern on negative edge
//     Enc/Outputs/Out/nCtrl1 @bit 1 <-> ENC Control compact/Control/Enable latch extern on positive edge
//     Enc/Outputs/Out/nCtrl1 @bit 2 <-> ENC Control compact/Control/Set counter
//     Enc/Outputs/Out/nDataOut1[0] <-> ENC Control compact/Set counter value
//   (this object) <-> Device 1 (EtherCAT)/Power (EK1200)/PLC Junction 2 (EK1122)/PLC Coupler 2 (EK1100)/PLC Junction 9 (EK1122)/X2 SL2K4-SCATTER/SL2K4-EL7031-E1
//     Drive/Inputs/In/nState1 @bit 3 <-> STM Status/Status/Error
//     Drive/Inputs/In/nState1 @bit 5 <-> STM Status/Status/Moving negative
//     Drive/Inputs/In/nState1 @bit 4 <-> STM Status/Status/Moving positive
//     Drive/Inputs/In/nState1 @bit 1 <-> STM Status/Status/Ready
//     Drive/Inputs/In/nState1 <-> STM Status/Status/Ready to enable
//     Drive/Inputs/In/nState1 @bit 6 <-> STM Status/Status/Torque reduced
//     Drive/Inputs/In/nState1 @bit 2 <-> STM Status/Status/Warning
//     Drive/Inputs/In/nState2 @bit 3 <-> STM Status/Status/Digital input 1
//     Drive/Inputs/In/nState2 @bit 4 <-> STM Status/Status/Digital input 2
//     Drive/Inputs/In/nState2 @bit 5 <-> STM Status/Status/Sync error
//     Drive/Inputs/In/nState2 @bit 7 <-> STM Status/Status/TxPDO Toggle
//     Drive/Inputs/In/nState4 @bit 1 <-> WcState/InputToggle
//     Drive/Inputs/In/nState4 <-> WcState/WcState
//     Drive/Outputs/Out/nCtrl1 <-> STM Control/Control/Enable
//     Drive/Outputs/Out/nCtrl1 @bit 2 <-> STM Control/Control/Reduce torque
//     Drive/Outputs/Out/nCtrl1 @bit 1 <-> STM Control/Control/Reset
//     Drive/Outputs/Out/nDataOut2[0] <-> STM Velocity/Velocity
//   (this object) <-> Device 1 (EtherCAT)/Power (EK1200)/PLC Junction 2 (EK1122)/PLC Coupler 2 (EK1100)/PLC Junction 9 (EK1122)/X2 SL2K4-SCATTER/SL2K4-EL5101-E4
//     Enc/Inputs/In/nDataIn1[0] <-> ENC Status compact/Counter value
//     Enc/Inputs/In/nDataIn2[0] <-> ENC Status compact/Latch value
//     Enc/Inputs/In/nState1 @bit 4 <-> ENC Status compact/Status/Counter overflow
//     Enc/Inputs/In/nState1 @bit 3 <-> ENC Status compact/Status/Counter underflow
//     Enc/Inputs/In/nState1 @bit 7 <-> ENC Status compact/Status/Extrapolation stall
//     Enc/Inputs/In/nState1 <-> ENC Status compact/Status/Latch C valid
//     Enc/Inputs/In/nState1 @bit 1 <-> ENC Status compact/Status/Latch extern valid
//     Enc/Inputs/In/nState1 @bit 6 <-> ENC Status compact/Status/Open circuit
//     Enc/Inputs/In/nState1 @bit 2 <-> ENC Status compact/Status/Set counter done
//     Enc/Inputs/In/nState1 @bit 5 <-> ENC Status compact/Status/Status of input status
//     Enc/Inputs/In/nState2 @bit 4 <-> ENC Status compact/Status/Status of extern latch
//     Enc/Inputs/In/nState2 <-> ENC Status compact/Status/Status of input A
//     Enc/Inputs/In/nState2 @bit 1 <-> ENC Status compact/Status/Status of input B
//     Enc/Inputs/In/nState2 @bit 2 <-> ENC Status compact/Status/Status of input C
//     Enc/Inputs/In/nState2 @bit 3 <-> ENC Status compact/Status/Status of input gate
//     Enc/Inputs/In/nState2 @bit 5 <-> ENC Status compact/Status/Sync error
//     Enc/Inputs/In/nState2 @bit 6 <-> ENC Status compact/Status/TxPDO State
//     Enc/Inputs/In/nState2 @bit 7 <-> ENC Status compact/Status/TxPDO Toggle
//     Enc/Inputs/In/nState4 @bit 1 <-> WcState/InputToggle
//     Enc/Inputs/In/nState4 <-> WcState/WcState
//     Enc/Outputs/Out/nCtrl1 <-> ENC Control compact/Control/Enable latch C
//     Enc/Outputs/Out/nCtrl1 @bit 3 <-> ENC Control compact/Control/Enable latch extern on negative edge
//     Enc/Outputs/Out/nCtrl1 @bit 1 <-> ENC Control compact/Control/Enable latch extern on positive edge
//     Enc/Outputs/Out/nCtrl1 @bit 2 <-> ENC Control compact/Control/Set counter
//     Enc/Outputs/Out/nDataOut1[0] <-> ENC Control compact/Set counter value
//   (this object) <-> Device 1 (EtherCAT)/Power (EK1200)/PLC Junction 2 (EK1122)/PLC Coupler 2 (EK1100)/PLC Junction 9 (EK1122)/X2 SL2K4-SCATTER/SL2K4-EL7031-E3
//     Drive/Inputs/In/nState1 @bit 3 <-> STM Status/Status/Error
//     Drive/Inputs/In/nState1 @bit 5 <-> STM Status/Status/Moving negative
//     Drive/Inputs/In/nState1 @bit 4 <-> STM Status/Status/Moving positive
//     Drive/Inputs/In/nState1 @bit 1 <-> STM Status/Status/Ready
//     Drive/Inputs/In/nState1 <-> STM Status/Status/Ready to enable
//     Drive/Inputs/In/nState1 @bit 6 <-> STM Status/Status/Torque reduced
//     Drive/Inputs/In/nState1 @bit 2 <-> STM Status/Status/Warning
//     Drive/Inputs/In/nState2 @bit 3 <-> STM Status/Status/Digital input 1
//     Drive/Inputs/In/nState2 @bit 4 <-> STM Status/Status/Digital input 2
//     Drive/Inputs/In/nState2 @bit 5 <-> STM Status/Status/Sync error
//     Drive/Inputs/In/nState2 @bit 7 <-> STM Status/Status/TxPDO Toggle
//     Drive/Inputs/In/nState4 @bit 1 <-> WcState/InputToggle
//     Drive/Inputs/In/nState4 <-> WcState/WcState
//     Drive/Outputs/Out/nCtrl1 <-> STM Control/Control/Enable
//     Drive/Outputs/Out/nCtrl1 @bit 2 <-> STM Control/Control/Reduce torque
//     Drive/Outputs/Out/nCtrl1 @bit 1 <-> STM Control/Control/Reset
//     Drive/Outputs/Out/nDataOut2[0] <-> STM Velocity/Velocity
//   (this object) <-> Device 1 (EtherCAT)/Power (EK1200)/PLC Junction 2 (EK1122)/PLC Coupler 2 (EK1100)/PLC Junction 9 (EK1122)/X2 SL2K4-SCATTER/SL2K4-EL5101-E6
//     Enc/Inputs/In/nDataIn1[0] <-> ENC Status compact/Counter value
//     Enc/Inputs/In/nDataIn2[0] <-> ENC Status compact/Latch value
//     Enc/Inputs/In/nState1 @bit 4 <-> ENC Status compact/Status/Counter overflow
//     Enc/Inputs/In/nState1 @bit 3 <-> ENC Status compact/Status/Counter underflow
//     Enc/Inputs/In/nState1 @bit 7 <-> ENC Status compact/Status/Extrapolation stall
//     Enc/Inputs/In/nState1 <-> ENC Status compact/Status/Latch C valid
//     Enc/Inputs/In/nState1 @bit 1 <-> ENC Status compact/Status/Latch extern valid
//     Enc/Inputs/In/nState1 @bit 6 <-> ENC Status compact/Status/Open circuit
//     Enc/Inputs/In/nState1 @bit 2 <-> ENC Status compact/Status/Set counter done
//     Enc/Inputs/In/nState1 @bit 5 <-> ENC Status compact/Status/Status of input status
//     Enc/Inputs/In/nState2 @bit 4 <-> ENC Status compact/Status/Status of extern latch
//     Enc/Inputs/In/nState2 <-> ENC Status compact/Status/Status of input A
//     Enc/Inputs/In/nState2 @bit 1 <-> ENC Status compact/Status/Status of input B
//     Enc/Inputs/In/nState2 @bit 2 <-> ENC Status compact/Status/Status of input C
//     Enc/Inputs/In/nState2 @bit 3 <-> ENC Status compact/Status/Status of input gate
//     Enc/Inputs/In/nState2 @bit 5 <-> ENC Status compact/Status/Sync error
//     Enc/Inputs/In/nState2 @bit 6 <-> ENC Status compact/Status/TxPDO State
//     Enc/Inputs/In/nState2 @bit 7 <-> ENC Status compact/Status/TxPDO Toggle
//     Enc/Inputs/In/nState4 @bit 1 <-> WcState/InputToggle
//     Enc/Inputs/In/nState4 <-> WcState/WcState
//     Enc/Outputs/Out/nCtrl1 <-> ENC Control compact/Control/Enable latch C
//     Enc/Outputs/Out/nCtrl1 @bit 3 <-> ENC Control compact/Control/Enable latch extern on negative edge
//     Enc/Outputs/Out/nCtrl1 @bit 1 <-> ENC Control compact/Control/Enable latch extern on positive edge
//     Enc/Outputs/Out/nCtrl1 @bit 2 <-> ENC Control compact/Control/Set counter
//     Enc/Outputs/Out/nDataOut1[0] <-> ENC Control compact/Set counter value
//   (this object) <-> Device 1 (EtherCAT)/Power (EK1200)/PLC Junction 2 (EK1122)/PLC Coupler 2 (EK1100)/PLC Junction 9 (EK1122)/X2 SL2K4-SCATTER/SL2K4-EL7031-E5
//     Drive/Inputs/In/nState1 @bit 3 <-> STM Status/Status/Error
//     Drive/Inputs/In/nState1 @bit 5 <-> STM Status/Status/Moving negative
//     Drive/Inputs/In/nState1 @bit 4 <-> STM Status/Status/Moving positive
//     Drive/Inputs/In/nState1 @bit 1 <-> STM Status/Status/Ready
//     Drive/Inputs/In/nState1 <-> STM Status/Status/Ready to enable
//     Drive/Inputs/In/nState1 @bit 6 <-> STM Status/Status/Torque reduced
//     Drive/Inputs/In/nState1 @bit 2 <-> STM Status/Status/Warning
//     Drive/Inputs/In/nState2 @bit 3 <-> STM Status/Status/Digital input 1
//     Drive/Inputs/In/nState2 @bit 4 <-> STM Status/Status/Digital input 2
//     Drive/Inputs/In/nState2 @bit 5 <-> STM Status/Status/Sync error
//     Drive/Inputs/In/nState2 @bit 7 <-> STM Status/Status/TxPDO Toggle
//     Drive/Inputs/In/nState4 @bit 1 <-> WcState/InputToggle
//     Drive/Inputs/In/nState4 <-> WcState/WcState
//     Drive/Outputs/Out/nCtrl1 <-> STM Control/Control/Enable
//     Drive/Outputs/Out/nCtrl1 @bit 2 <-> STM Control/Control/Reduce torque
//     Drive/Outputs/Out/nCtrl1 @bit 1 <-> STM Control/Control/Reset
//     Drive/Outputs/Out/nDataOut2[0] <-> STM Velocity/Velocity
//   (this object) <-> Device 1 (EtherCAT)/Power (EK1200)/PLC Junction 2 (EK1122)/PLC Coupler 2 (EK1100)/PLC Junction 9 (EK1122)/X2 SL2K4-SCATTER/SL2K4-EL5101-E8
//     Enc/Inputs/In/nDataIn1[0] <-> ENC Status compact/Counter value
//     Enc/Inputs/In/nDataIn2[0] <-> ENC Status compact/Latch value
//     Enc/Inputs/In/nState1 @bit 4 <-> ENC Status compact/Status/Counter overflow
//     Enc/Inputs/In/nState1 @bit 3 <-> ENC Status compact/Status/Counter underflow
//     Enc/Inputs/In/nState1 @bit 7 <-> ENC Status compact/Status/Extrapolation stall
//     Enc/Inputs/In/nState1 <-> ENC Status compact/Status/Latch C valid
//     Enc/Inputs/In/nState1 @bit 1 <-> ENC Status compact/Status/Latch extern valid
//     Enc/Inputs/In/nState1 @bit 6 <-> ENC Status compact/Status/Open circuit
//     Enc/Inputs/In/nState1 @bit 2 <-> ENC Status compact/Status/Set counter done
//     Enc/Inputs/In/nState1 @bit 5 <-> ENC Status compact/Status/Status of input status
//     Enc/Inputs/In/nState2 @bit 4 <-> ENC Status compact/Status/Status of extern latch
//     Enc/Inputs/In/nState2 <-> ENC Status compact/Status/Status of input A
//     Enc/Inputs/In/nState2 @bit 1 <-> ENC Status compact/Status/Status of input B
//     Enc/Inputs/In/nState2 @bit 2 <-> ENC Status compact/Status/Status of input C
//     Enc/Inputs/In/nState2 @bit 3 <-> ENC Status compact/Status/Status of input gate
//     Enc/Inputs/In/nState2 @bit 5 <-> ENC Status compact/Status/Sync error
//     Enc/Inputs/In/nState2 @bit 6 <-> ENC Status compact/Status/TxPDO State
//     Enc/Inputs/In/nState2 @bit 7 <-> ENC Status compact/Status/TxPDO Toggle
//     Enc/Inputs/In/nState4 @bit 1 <-> WcState/InputToggle
//     Enc/Inputs/In/nState4 <-> WcState/WcState
//     Enc/Outputs/Out/nCtrl1 <-> ENC Control compact/Control/Enable latch C
//     Enc/Outputs/Out/nCtrl1 @bit 3 <-> ENC Control compact/Control/Enable latch extern on negative edge
//     Enc/Outputs/Out/nCtrl1 @bit 1 <-> ENC Control compact/Control/Enable latch extern on positive edge
//     Enc/Outputs/Out/nCtrl1 @bit 2 <-> ENC Control compact/Control/Set counter
//     Enc/Outputs/Out/nDataOut1[0] <-> ENC Control compact/Set counter value
//   (this object) <-> Device 1 (EtherCAT)/Power (EK1200)/PLC Junction 2 (EK1122)/PLC Coupler 2 (EK1100)/PLC Junction 9 (EK1122)/X2 SL2K4-SCATTER/SL2K4-EL7031-E7
//     Drive/Inputs/In/nState1 @bit 3 <-> STM Status/Status/Error
//     Drive/Inputs/In/nState1 @bit 5 <-> STM Status/Status/Moving negative
//     Drive/Inputs/In/nState1 @bit 4 <-> STM Status/Status/Moving positive
//     Drive/Inputs/In/nState1 @bit 1 <-> STM Status/Status/Ready
//     Drive/Inputs/In/nState1 <-> STM Status/Status/Ready to enable
//     Drive/Inputs/In/nState1 @bit 6 <-> STM Status/Status/Torque reduced
//     Drive/Inputs/In/nState1 @bit 2 <-> STM Status/Status/Warning
//     Drive/Inputs/In/nState2 @bit 3 <-> STM Status/Status/Digital input 1
//     Drive/Inputs/In/nState2 @bit 4 <-> STM Status/Status/Digital input 2
//     Drive/Inputs/In/nState2 @bit 5 <-> STM Status/Status/Sync error
//     Drive/Inputs/In/nState2 @bit 7 <-> STM Status/Status/TxPDO Toggle
//     Drive/Inputs/In/nState4 @bit 1 <-> WcState/InputToggle
//     Drive/Inputs/In/nState4 <-> WcState/WcState
//     Drive/Outputs/Out/nCtrl1 <-> STM Control/Control/Enable
